gfCNCPoint2[19223] = {X 326.2725, Y 101.3575, Z -3.0000, A 0.000, B 0.000, C 0.000 }
gfCNCPoint2[19224] = {X 323.4288, Y 100.7538, Z -3.0000, A 0.000, B 0.000, C 0.000 }
gfCNCPoint2[19225] = {X 320.6373, Y 99.9425, Z -3.0000, A 0.000, B 0.000, C 0.000 }
gfCNCPoint2[19226] = {X 317.9129, Y 98.9281, Z -3.0000, A 0.000, B 0.000, C 0.000 }
gfCNCPoint2[19227] = {X 316.4064, Y 98.2325, Z -3.0000, A 0.000, B 0.000, C 0.000 }
gfCNCPoint2[19228] = {X 314.9630, Y 97.4138, Z -3.0000, A 0.000, B 0.000, C 0.000 }
gfCNCPoint2[19229] = {X 313.5930, Y 96.4776, Z -3.0000, A 0.000, B 0.000, C 0.000 }
gfCNCPoint2[19230] = {X 312.3057, Y 95.4305, Z -3.0000, A 0.000, B 0.000, C 0.000 }
gfCNCPoint2[19231] = {X 311.3087, Y 94.4389, Z -3.0000, A 0.000, B 0.000, C 0.000 }
gfCNCPoint2[19232] = {X 310.4363, Y 93.3361, Z -3.0000, A 0.000, B 0.000, C 0.000 }
gfCNCPoint2[19233] = {X 309.7010, Y 92.1376, Z -3.0000, A 0.000, B 0.000, C 0.000 }
gfCNCPoint2[19234] = {X 309.1130, Y 90.8602, Z -3.0000, A 0.000, B 0.000, C 0.000 }
gfCNCPoint2[19235] = {X 308.6807, Y 89.5222, Z -3.0000, A 0.000, B 0.000, C 0.000 }
gfCNCPoint2[19236] = {X 308.3387, Y 87.9058, Z -3.0000, A 0.000, B 0.000, C 0.000 }
gfCNCPoint2[19237] = {X 308.1366, Y 86.2660, Z -3.0000, A 0.000, B 0.000, C 0.000 }
gfCNCPoint2[19238] = {X 308.0760, Y 84.6149, Z -3.0000, A 0.000, B 0.000, C 0.000 }
gfCNCPoint2[19239] = {X 308.0773, Y 83.2310, Z -3.0000, A 0.000, B 0.000, C 0.000 }
gfCNCPoint2[19240] = {X 308.0773, Y 63.1422, Z -3.0000, A 0.000, B 0.000, C 0.000 }
gfCNCPoint2[19241] = {X 307.2288, Y 62.9475, Z -3.0000, A 0.000, B 0.000, C 0.000 }
gfCNCPoint2[19242] = {X 306.4379, Y 62.5836, Z -3.0000, A 0.000, B 0.000, C 0.000 }
gfCNCPoint2[19243] = {X 305.7380, Y 62.0658, Z -3.0000, A 0.000, B 0.000, C 0.000 }
gfCNCPoint2[19244] = {X 305.1586, Y 61.4160, Z -3.0000, A 0.000, B 0.000, C 0.000 }
gfCNCPoint2[19245] = {X 304.7241, Y 60.6616, Z -3.0000, A 0.000, B 0.000, C 0.000 }
gfCNCPoint2[19246] = {X 304.4529, Y 59.8343, Z -3.0000, A 0.000, B 0.000, C 0.000 }
gfCNCPoint2[19247] = {X 304.3564, Y 58.9691, Z -3.0000, A 0.000, B 0.000, C 0.000 }
gfCNCPoint2[19248] = {X 304.3562, Y 58.0000, Z -3.0000, A 0.000, B 0.000, C 0.000 }
gfCNCPoint2[19249] = {X 304.4625, Y 57.0565, Z -3.0000, A 0.000, B 0.000, C 0.000 }
gfCNCPoint2[19250] = {X 304.7761, Y 56.1603, Z -3.0000, A 0.000, B 0.000, C 0.000 }
gfCNCPoint2[19251] = {X 305.2813, Y 55.3564, Z -3.0000, A 0.000, B 0.000, C 0.000 }
gfCNCPoint2[19252] = {X 305.9526, Y 54.6850, Z -3.0000, A 0.000, B 0.000, C 0.000 }
gfCNCPoint2[19253] = {X 306.7566, Y 54.1799, Z -3.0000, A 0.000, B 0.000, C 0.000 }
gfCNCPoint2[19254] = {X 307.6527, Y 53.8663, Z -3.0000, A 0.000, B 0.000, C 0.000 }
gfCNCPoint2[19255] = {X 308.5962, Y 53.7600, Z -3.0000, A 0.000, B 0.000, C 0.000 }
gfCNCPoint2[19256] = {X 324.3107, Y 53.7600, Z -3.0000, A 0.000, B 0.000, C 0.000 }
gfCNCPoint2[19257] = {X 325.2542, Y 53.8663, Z -3.0000, A 0.000, B 0.000, C 0.000 }
gfCNCPoint2[19258] = {X 326.1504, Y 54.1799, Z -3.0000, A 0.000, B 0.000, C 0.000 }
gfCNCPoint2[19259] = {X 326.9543, Y 54.6850, Z -3.0000, A 0.000, B 0.000, C 0.000 }
gfCNCPoint2[19260] = {X 327.6257, Y 55.3564, Z -3.0000, A 0.000, B 0.000, C 0.000 }
gfCNCPoint2[19261] = {X 328.1308, Y 56.1603, Z -3.0000, A 0.000, B 0.000, C 0.000 }
gfCNCPoint2[19262] = {X 328.4444, Y 57.0565, Z -3.0000, A 0.000, B 0.000, C 0.000 }
gfCNCPoint2[19263] = {X 328.5507, Y 58.0000, Z -3.0000, A 0.000, B 0.000, C 0.000 }
gfCNCPoint2[19264] = {X 328.5507, Y 58.9355, Z -3.0000, A 0.000, B 0.000, C 0.000 }
gfCNCPoint2[19265] = {X 328.4560, Y 59.8053, Z -3.0000, A 0.000, B 0.000, C 0.000 }
gfCNCPoint2[19266] = {X 328.1864, Y 60.6376, Z -3.0000, A 0.000, B 0.000, C 0.000 }
gfCNCPoint2[19267] = {X 327.7532, Y 61.3977, Z -3.0000, A 0.000, B 0.000, C 0.000 }
gfCNCPoint2[19268] = {X 327.1745, Y 62.0538, Z -3.0000, A 0.000, B 0.000, C 0.000 }
gfCNCPoint2[19269] = {X 326.4744, Y 62.5785, Z -3.0000, A 0.000, B 0.000, C 0.000 }
gfCNCPoint2[19270] = {X 325.6822, Y 62.9499, Z -3.0000, A 0.000, B 0.000, C 0.000 }
gfCNCPoint2[19271] = {X 324.8311, Y 63.1523, Z -3.0000, A 0.000, B 0.000, C 0.000 }
gfCNCPoint2[19272] = {X 324.8326, Y 83.2300, Z -3.0000, A 0.000, B 0.000, C 0.000 }
gfCNCPoint2[19273] = {X 324.8461, Y 84.6151, Z -3.0000, A 0.000, B 0.000, C 0.000 }
gfCNCPoint2[19274] = {X 324.9250, Y 85.8673, Z -3.0000, A 0.000, B 0.000, C 0.000 }
gfCNCPoint2[19275] = {X 325.1520, Y 87.1014, Z -3.0000, A 0.000, B 0.000, C 0.000 }
gfCNCPoint2[19276] = {X 325.4127, Y 87.3915, Z -3.0000, A 0.000, B 0.000, C 0.000 }
gfCNCPoint2[19277] = {X 325.7358, Y 87.6100, Z -3.0000, A 0.000, B 0.000, C 0.000 }
gfCNCPoint2[19278] = {X 326.1869, Y 87.8647, Z -3.0000, A 0.000, B 0.000, C 0.000 }
gfCNCPoint2[19279] = {X 327.6340, Y 88.4662, Z -3.0000, A 0.000, B 0.000, C 0.000 }
gfCNCPoint2[19280] = {X 329.1387, Y 88.9046, Z -3.0000, A 0.000, B 0.000, C 0.000 }
gfCNCPoint2[19281] = {X 332.2202, Y 89.5215, Z -3.0000, A 0.000, B 0.000, C 0.000 }
gfCNCPoint2[19282] = {X 335.3381, Y 89.9149, Z -3.0000, A 0.000, B 0.000, C 0.000 }
gfCNCPoint2[19283] = {X 339.4788, Y 90.2356, Z -3.0000, A 0.000, B 0.000, C 0.000 }
gfCNCPoint2[19284] = {X 343.6280, Y 90.4154, Z -3.0000, A 0.000, B 0.000, C 0.000 }
gfCNCPoint2[19285] = {X 347.7809, Y 90.4540, Z -3.0000, A 0.000, B 0.000, C 0.000 }
gfCNCPoint2[19286] = {X 352.1650, Y 90.4156, Z -3.0000, A 0.000, B 0.000, C 0.000 }
gfCNCPoint2[19287] = {X 356.5449, Y 90.2196, Z -3.0000, A 0.000, B 0.000, C 0.000 }
gfCNCPoint2[19288] = {X 360.9150, Y 89.8663, Z -3.0000, A 0.000, B 0.000, C 0.000 }
gfCNCPoint2[19289] = {X 363.2338, Y 89.5779, Z -3.0000, A 0.000, B 0.000, C 0.000 }
gfCNCPoint2[19290] = {X 365.5310, Y 89.1507, Z -3.0000, A 0.000, B 0.000, C 0.000 }
gfCNCPoint2[19291] = {X 367.7985, Y 88.5862, Z -3.0000, A 0.000, B 0.000, C 0.000 }
gfCNCPoint2[19292] = {X 368.7389, Y 88.2700, Z -3.0000, A 0.000, B 0.000, C 0.000 }
gfCNCPoint2[19293] = {X 369.6379, Y 87.8503, Z -3.0000, A 0.000, B 0.000, C 0.000 }
gfCNCPoint2[19294] = {X 370.4842, Y 87.3325, Z -3.0000, A 0.000, B 0.000, C 0.000 }
gfCNCPoint2[19295] = {X 370.6562, Y 87.1535, Z -3.0000, A 0.000, B 0.000, C 0.000 }
gfCNCPoint2[19296] = {X 370.7448, Y 86.9218, Z -3.0000, A 0.000, B 0.000, C 0.000 }
gfCNCPoint2[19297] = {X 370.9367, Y 85.3801, Z -3.0000, A 0.000, B 0.000, C 0.000 }
gfCNCPoint2[19298] = {X 371.0008, Y 83.8280, Z -3.0000, A 0.000, B 0.000, C 0.000 }
gfCNCPoint2[19299] = {X 371.0008, Y 63.1422, Z -3.0000, A 0.000, B 0.000, C 0.000 }
gfCNCPoint2[19300] = {X 370.1522, Y 62.9476, Z -3.0000, A 0.000, B 0.000, C 0.000 }
gfCNCPoint2[19301] = {X 369.3612, Y 62.5838, Z -3.0000, A 0.000, B 0.000, C 0.000 }
gfCNCPoint2[19302] = {X 368.6612, Y 62.0660, Z -3.0000, A 0.000, B 0.000, C 0.000 }
gfCNCPoint2[19303] = {X 368.0817, Y 61.4162, Z -3.0000, A 0.000, B 0.000, C 0.000 }
gfCNCPoint2[19304] = {X 367.6472, Y 60.6617, Z -3.0000, A 0.000, B 0.000, C 0.000 }
gfCNCPoint2[19305] = {X 367.3760, Y 59.8344, Z -3.0000, A 0.000, B 0.000, C 0.000 }
gfCNCPoint2[19306] = {X 367.2794, Y 58.9691, Z -3.0000, A 0.000, B 0.000, C 0.000 }
gfCNCPoint2[19307] = {X 367.2793, Y 58.0000, Z -3.0000, A 0.000, B 0.000, C 0.000 }
gfCNCPoint2[19308] = {X 367.3856, Y 57.0565, Z -3.0000, A 0.000, B 0.000, C 0.000 }
gfCNCPoint2[19309] = {X 367.6992, Y 56.1603, Z -3.0000, A 0.000, B 0.000, C 0.000 }
gfCNCPoint2[19310] = {X 368.2043, Y 55.3564, Z -3.0000, A 0.000, B 0.000, C 0.000 }
gfCNCPoint2[19311] = {X 368.8757, Y 54.6850, Z -3.0000, A 0.000, B 0.000, C 0.000 }
gfCNCPoint2[19312] = {X 369.6796, Y 54.1799, Z -3.0000, A 0.000, B 0.000, C 0.000 }
gfCNCPoint2[19313] = {X 370.5758, Y 53.8663, Z -3.0000, A 0.000, B 0.000, C 0.000 }
gfCNCPoint2[19314] = {X 371.5193, Y 53.7600, Z -3.0000, A 0.000, B 0.000, C 0.000 }
gfCNCPoint2[19315] = {X 388.0597, Y 53.7600, Z -3.0000, A 0.000, B 0.000, C 0.000 }
gfCNCPoint2[19316] = {X 389.0032, Y 53.8663, Z -3.0000, A 0.000, B 0.000, C 0.000 }
gfCNCPoint2[19317] = {X 389.8993, Y 54.1799, Z -3.0000, A 0.000, B 0.000, C 0.000 }
gfCNCPoint2[19318] = {X 390.7033, Y 54.6850, Z -3.0000, A 0.000, B 0.000, C 0.000 }
gfCNCPoint2[19319] = {X 391.3746, Y 55.3564, Z -3.0000, A 0.000, B 0.000, C 0.000 }
gfCNCPoint2[19320] = {X 391.8798, Y 56.1603, Z -3.0000, A 0.000, B 0.000, C 0.000 }
gfCNCPoint2[19321] = {X 392.1934, Y 57.0565, Z -3.0000, A 0.000, B 0.000, C 0.000 }
gfCNCPoint2[19322] = {X 392.2997, Y 58.0000, Z -3.0000, A 0.000, B 0.000, C 0.000 }
gfCNCPoint2[19323] = {X 392.2997, Y 58.9342, Z -3.0000, A 0.000, B 0.000, C 0.000 }
gfCNCPoint2[19324] = {X 392.1866, Y 59.9066, Z -3.0000, A 0.000, B 0.000, C 0.000 }
gfCNCPoint2[19325] = {X 391.8536, Y 60.8272, Z -3.0000, A 0.000, B 0.000, C 0.000 }
gfCNCPoint2[19326] = {X 391.4098, Y 61.5353, Z -3.0000, A 0.000, B 0.000, C 0.000 }
gfCNCPoint2[19327] = {X 390.8364, Y 62.1431, Z -3.0000, A 0.000, B 0.000, C 0.000 }
gfCNCPoint2[19328] = {X 390.1553, Y 62.6274, Z -3.0000, A 0.000, B 0.000, C 0.000 }
gfCNCPoint2[19329] = {X 389.3929, Y 62.9695, Z -3.0000, A 0.000, B 0.000, C 0.000 }
gfCNCPoint2[19330] = {X 388.5783, Y 63.1561, Z -3.0000, A 0.000, B 0.000, C 0.000 }
gfCNCPoint2[19331] = {X 388.5763, Y 84.6150, Z -3.0000, A 0.000, B 0.000, C 0.000 }
gfCNCPoint2[19332] = {X 388.5167, Y 86.2665, Z -3.0000, A 0.000, B 0.000, C 0.000 }
gfCNCPoint2[19333] = {X 388.3133, Y 87.9065, Z -3.0000, A 0.000, B 0.000, C 0.000 }
gfCNCPoint2[19334] = {X 387.9674, Y 89.5225, Z -3.0000, A 0.000, B 0.000, C 0.000 }
gfCNCPoint2[19335] = {X 387.4388, Y 91.0992, Z -3.0000, A 0.000, B 0.000, C 0.000 }
gfCNCPoint2[19336] = {X 386.6944, Y 92.5861, Z -3.0000, A 0.000, B 0.000, C 0.000 }
gfCNCPoint2[19337] = {X 385.7486, Y 93.9539, Z -3.0000, A 0.000, B 0.000, C 0.000 }
gfCNCPoint2[19338] = {X 384.6203, Y 95.1755, Z -3.0000, A 0.000, B 0.000, C 0.000 }
gfCNCPoint2[19339] = {X 383.1126, Y 96.4458, Z -3.0000, A 0.000, B 0.000, C 0.000 }
gfCNCPoint2[19340] = {X 381.4786, Y 97.5489, Z -3.0000, A 0.000, B 0.000, C 0.000 }
gfCNCPoint2[19341] = {X 379.7367, Y 98.4723, Z -3.0000, A 0.000, B 0.000, C 0.000 }
gfCNCPoint2[19342] = {X 377.4708, Y 99.4262, Z -3.0000, A 0.000, B 0.000, C 0.000 }
gfCNCPoint2[19343] = {X 375.1422, Y 100.2147, Z -3.0000, A 0.000, B 0.000, C 0.000 }
gfCNCPoint2[19344] = {X 372.7628, Y 100.8335, Z -3.0000, A 0.000, B 0.000, C 0.000 }
gfCNCPoint2[19345] = {X 368.9550, Y 101.5702, Z -3.0000, A 0.000, B 0.000, C 0.000 }
gfCNCPoint2[19346] = {X 365.1161, Y 102.1230, Z -3.0000, A 0.000, B 0.000, C 0.000 }
gfCNCPoint2[19347] = {X 361.2551, Y 102.4906, Z -3.0000, A 0.000, B 0.000, C 0.000 }
gfCNCPoint2[19348] = {X 357.2498, Y 102.7312, Z -3.0000, A 0.000, B 0.000, C 0.000 }
gfCNCPoint2[19349] = {X 353.2403, Y 102.8846, Z -3.0000, A 0.000, B 0.000, C 0.000 }
gfCNCPoint2[19350] = {X 353.3497, Y 106.8831, Z -3.0000, A 0.000, B 0.000, C 0.000 }
gfCNCPoint2[19351] = {X 353.2381, Y 102.8046, Z -3.0000, A 0.000, B 0.000, C 0.000 }
gfCNCPoint2[19352] = {X 347.7206, Y 102.8731, Z -3.0000, A 0.000, B 0.000, C 0.000 }
gfCNCPoint2[19353] = {X 342.2035, Y 102.7764, Z -3.0000, A 0.000, B 0.000, C 0.000 }
gfCNCPoint2[19354] = {X 336.6917, Y 102.5147, Z -3.0000, A 0.000, B 0.000, C 0.000 }
gfCNCPoint2[19355] = {X 333.2080, Y 102.2391, Z -3.0000, A 0.000, B 0.000, C 0.000 }
gfCNCPoint2[19356] = {X 329.7378, Y 101.8269, Z -3.0000, A 0.000, B 0.000, C 0.000 }
gfCNCPoint2[19357] = {X 326.2865, Y 101.2787, Z -3.0000, A 0.000, B 0.000, C 0.000 }
gfCNCPoint2[19358] = {X 323.4485, Y 100.6762, Z -3.0000, A 0.000, B 0.000, C 0.000 }
gfCNCPoint2[19359] = {X 320.6624, Y 99.8666, Z -3.0000, A 0.000, B 0.000, C 0.000 }
gfCNCPoint2[19360] = {X 317.9435, Y 98.8541, Z -3.0000, A 0.000, B 0.000, C 0.000 }
gfCNCPoint2[19361] = {X 316.4430, Y 98.1614, Z -3.0000, A 0.000, B 0.000, C 0.000 }
gfCNCPoint2[19362] = {X 315.0054, Y 97.3460, Z -3.0000, A 0.000, B 0.000, C 0.000 }
gfCNCPoint2[19363] = {X 313.6408, Y 96.4135, Z -3.0000, A 0.000, B 0.000, C 0.000 }
gfCNCPoint2[19364] = {X 312.3587, Y 95.3706, Z -3.0000, A 0.000, B 0.000, C 0.000 }
gfCNCPoint2[19365] = {X 311.3684, Y 94.3857, Z -3.0000, A 0.000, B 0.000, C 0.000 }
gfCNCPoint2[19366] = {X 310.5019, Y 93.2903, Z -3.0000, A 0.000, B 0.000, C 0.000 }
gfCNCPoint2[19367] = {X 309.7715, Y 92.0999, Z -3.0000, A 0.000, B 0.000, C 0.000 }
gfCNCPoint2[19368] = {X 309.1875, Y 90.8312, Z -3.0000, A 0.000, B 0.000, C 0.000 }
gfCNCPoint2[19369] = {X 308.7582, Y 89.5022, Z -3.0000, A 0.000, B 0.000, C 0.000 }
gfCNCPoint2[19370] = {X 308.4176, Y 87.8925, Z -3.0000, A 0.000, B 0.000, C 0.000 }
gfCNCPoint2[19371] = {X 308.2164, Y 86.2595, Z -3.0000, A 0.000, B 0.000, C 0.000 }
gfCNCPoint2[19372] = {X 308.1560, Y 84.6152, Z -3.0000, A 0.000, B 0.000, C 0.000 }
gfCNCPoint2[19373] = {X 308.1573, Y 83.2311, Z -3.0000, A 0.000, B 0.000, C 0.000 }
gfCNCPoint2[19374] = {X 308.1573, Y 63.0708, Z -3.0000, A 0.000, B 0.000, C 0.000 }
gfCNCPoint2[19375] = {X 307.3120, Y 62.8909, Z -3.0000, A 0.000, B 0.000, C 0.000 }
gfCNCPoint2[19376] = {X 306.5222, Y 62.5402, Z -3.0000, A 0.000, B 0.000, C 0.000 }
gfCNCPoint2[19377] = {X 305.8219, Y 62.0338, Z -3.0000, A 0.000, B 0.000, C 0.000 }
gfCNCPoint2[19378] = {X 305.2413, Y 61.3937, Z -3.0000, A 0.000, B 0.000, C 0.000 }
gfCNCPoint2[19379] = {X 304.8054, Y 60.6474, Z -3.0000, A 0.000, B 0.000, C 0.000 }
gfCNCPoint2[19380] = {X 304.5332, Y 59.8272, Z -3.0000, A 0.000, B 0.000, C 0.000 }
gfCNCPoint2[19381] = {X 304.4364, Y 58.9684, Z -3.0000, A 0.000, B 0.000, C 0.000 }
gfCNCPoint2[19382] = {X 304.4362, Y 58.0000, Z -3.0000, A 0.000, B 0.000, C 0.000 }
gfCNCPoint2[19383] = {X 304.5405, Y 57.0743, Z -3.0000, A 0.000, B 0.000, C 0.000 }
gfCNCPoint2[19384] = {X 304.8482, Y 56.1950, Z -3.0000, A 0.000, B 0.000, C 0.000 }
gfCNCPoint2[19385] = {X 305.3438, Y 55.4063, Z -3.0000, A 0.000, B 0.000, C 0.000 }
gfCNCPoint2[19386] = {X 306.0025, Y 54.7476, Z -3.0000, A 0.000, B 0.000, C 0.000 }
gfCNCPoint2[19387] = {X 306.7913, Y 54.2520, Z -3.0000, A 0.000, B 0.000, C 0.000 }
gfCNCPoint2[19388] = {X 307.6705, Y 53.9443, Z -3.0000, A 0.000, B 0.000, C 0.000 }
gfCNCPoint2[19389] = {X 308.5962, Y 53.8400, Z -3.0000, A 0.000, B 0.000, C 0.000 }
gfCNCPoint2[19390] = {X 324.3107, Y 53.8400, Z -3.0000, A 0.000, B 0.000, C 0.000 }
gfCNCPoint2[19391] = {X 325.2364, Y 53.9443, Z -3.0000, A 0.000, B 0.000, C 0.000 }
gfCNCPoint2[19392] = {X 326.1156, Y 54.2520, Z -3.0000, A 0.000, B 0.000, C 0.000 }
gfCNCPoint2[19393] = {X 326.9044, Y 54.7476, Z -3.0000, A 0.000, B 0.000, C 0.000 }
gfCNCPoint2[19394] = {X 327.5631, Y 55.4063, Z -3.0000, A 0.000, B 0.000, C 0.000 }
gfCNCPoint2[19395] = {X 328.0587, Y 56.1950, Z -3.0000, A 0.000, B 0.000, C 0.000 }
gfCNCPoint2[19396] = {X 328.3664, Y 57.0743, Z -3.0000, A 0.000, B 0.000, C 0.000 }
gfCNCPoint2[19397] = {X 328.4707, Y 58.0000, Z -3.0000, A 0.000, B 0.000, C 0.000 }
gfCNCPoint2[19398] = {X 328.4707, Y 58.9351, Z -3.0000, A 0.000, B 0.000, C 0.000 }
gfCNCPoint2[19399] = {X 328.3757, Y 59.7983, Z -3.0000, A 0.000, B 0.000, C 0.000 }
gfCNCPoint2[19400] = {X 328.1051, Y 60.6236, Z -3.0000, A 0.000, B 0.000, C 0.000 }
gfCNCPoint2[19401] = {X 327.6706, Y 61.3756, Z -3.0000, A 0.000, B 0.000, C 0.000 }
gfCNCPoint2[19402] = {X 327.0906, Y 62.0221, Z -3.0000, A 0.000, B 0.000, C 0.000 }
gfCNCPoint2[19403] = {X 326.3901, Y 62.5354, Z -3.0000, A 0.000, B 0.000, C 0.000 }
gfCNCPoint2[19404] = {X 325.5990, Y 62.8937, Z -3.0000, A 0.000, B 0.000, C 0.000 }
gfCNCPoint2[19405] = {X 324.7510, Y 63.0816, Z -3.0000, A 0.000, B 0.000, C 0.000 }
gfCNCPoint2[19406] = {X 324.7526, Y 83.2304, Z -3.0000, A 0.000, B 0.000, C 0.000 }
gfCNCPoint2[19407] = {X 324.7661, Y 84.6154, Z -3.0000, A 0.000, B 0.000, C 0.000 }
gfCNCPoint2[19408] = {X 324.8465, Y 85.8844, Z -3.0000, A 0.000, B 0.000, C 0.000 }
gfCNCPoint2[19409] = {X 325.0779, Y 87.1348, Z -3.0000, A 0.000, B 0.000, C 0.000 }
gfCNCPoint2[19410] = {X 325.3539, Y 87.4463, Z -3.0000, A 0.000, B 0.000, C 0.000 }
gfCNCPoint2[19411] = {X 325.6979, Y 87.6805, Z -3.0000, A 0.000, B 0.000, C 0.000 }
gfCNCPoint2[19412] = {X 326.1498, Y 87.9356, Z -3.0000, A 0.000, B 0.000, C 0.000 }
gfCNCPoint2[19413] = {X 327.6062, Y 88.5412, Z -3.0000, A 0.000, B 0.000, C 0.000 }
gfCNCPoint2[19414] = {X 329.1205, Y 88.9825, Z -3.0000, A 0.000, B 0.000, C 0.000 }
gfCNCPoint2[19415] = {X 332.2075, Y 89.6005, Z -3.0000, A 0.000, B 0.000, C 0.000 }
gfCNCPoint2[19416] = {X 335.3310, Y 89.9945, Z -3.0000, A 0.000, B 0.000, C 0.000 }
gfCNCPoint2[19417] = {X 339.4742, Y 90.3155, Z -3.0000, A 0.000, B 0.000, C 0.000 }
gfCNCPoint2[19418] = {X 343.6260, Y 90.4954, Z -3.0000, A 0.000, B 0.000, C 0.000 }
gfCNCPoint2[19419] = {X 347.7815, Y 90.5340, Z -3.0000, A 0.000, B 0.000, C 0.000 }
gfCNCPoint2[19420] = {X 352.1681, Y 90.4955, Z -3.0000, A 0.000, B 0.000, C 0.000 }
gfCNCPoint2[19421] = {X 356.5504, Y 90.2994, Z -3.0000, A 0.000, B 0.000, C 0.000 }
gfCNCPoint2[19422] = {X 360.9228, Y 89.9459, Z -3.0000, A 0.000, B 0.000, C 0.000 }
gfCNCPoint2[19423] = {X 363.2463, Y 89.6569, Z -3.0000, A 0.000, B 0.000, C 0.000 }
gfCNCPoint2[19424] = {X 365.5481, Y 89.2288, Z -3.0000, A 0.000, B 0.000, C 0.000 }
gfCNCPoint2[19425] = {X 367.8201, Y 88.6632, Z -3.0000, A 0.000, B 0.000, C 0.000 }
gfCNCPoint2[19426] = {X 368.7689, Y 88.3441, Z -3.0000, A 0.000, B 0.000, C 0.000 }
gfCNCPoint2[19427] = {X 369.6759, Y 87.9207, Z -3.0000, A 0.000, B 0.000, C 0.000 }
gfCNCPoint2[19428] = {X 370.5298, Y 87.3983, Z -3.0000, A 0.000, B 0.000, C 0.000 }
gfCNCPoint2[19429] = {X 370.7237, Y 87.1964, Z -3.0000, A 0.000, B 0.000, C 0.000 }
gfCNCPoint2[19430] = {X 370.8237, Y 86.9349, Z -3.0000, A 0.000, B 0.000, C 0.000 }
gfCNCPoint2[19431] = {X 371.0164, Y 85.3867, Z -3.0000, A 0.000, B 0.000, C 0.000 }
gfCNCPoint2[19432] = {X 371.0808, Y 83.8279, Z -3.0000, A 0.000, B 0.000, C 0.000 }
gfCNCPoint2[19433] = {X 371.0808, Y 63.0709, Z -3.0000, A 0.000, B 0.000, C 0.000 }
gfCNCPoint2[19434] = {X 370.9784, Y 63.0587, Z -3.0000, A 0.000, B 0.000, C 0.000 }
gfCNCPoint2[19435] = {X 370.8762, Y 63.0441, Z -3.0000, A 0.000, B 0.000, C 0.000 }
gfCNCPoint2[19436] = {X 369.9386, Y 62.7821, Z -3.0000, A 0.000, B 0.000, C 0.000 }
gfCNCPoint2[19437] = {X 369.0876, Y 62.3093, Z -3.0000, A 0.000, B 0.000, C 0.000 }
gfCNCPoint2[19438] = {X 368.3697, Y 61.6518, Z -3.0000, A 0.000, B 0.000, C 0.000 }
gfCNCPoint2[19439] = {X 367.8243, Y 60.8454, Z -3.0000, A 0.000, B 0.000, C 0.000 }
gfCNCPoint2[19440] = {X 367.4813, Y 59.9343, Z -3.0000, A 0.000, B 0.000, C 0.000 }
gfCNCPoint2[19441] = {X 367.3594, Y 58.9684, Z -3.0000, A 0.000, B 0.000, C 0.000 }
gfCNCPoint2[19442] = {X 367.3593, Y 58.0000, Z -3.0000, A 0.000, B 0.000, C 0.000 }
gfCNCPoint2[19443] = {X 367.4636, Y 57.0743, Z -3.0000, A 0.000, B 0.000, C 0.000 }
gfCNCPoint2[19444] = {X 367.7713, Y 56.1950, Z -3.0000, A 0.000, B 0.000, C 0.000 }
gfCNCPoint2[19445] = {X 368.2669, Y 55.4063, Z -3.0000, A 0.000, B 0.000, C 0.000 }
gfCNCPoint2[19446] = {X 368.9256, Y 54.7476, Z -3.0000, A 0.000, B 0.000, C 0.000 }
gfCNCPoint2[19447] = {X 369.7143, Y 54.2520, Z -3.0000, A 0.000, B 0.000, C 0.000 }
gfCNCPoint2[19448] = {X 370.5936, Y 53.9443, Z -3.0000, A 0.000, B 0.000, C 0.000 }
gfCNCPoint2[19449] = {X 371.5193, Y 53.8400, Z -3.0000, A 0.000, B 0.000, C 0.000 }
gfCNCPoint2[19450] = {X 388.0597, Y 53.8400, Z -3.0000, A 0.000, B 0.000, C 0.000 }
gfCNCPoint2[19451] = {X 388.9854, Y 53.9443, Z -3.0000, A 0.000, B 0.000, C 0.000 }
gfCNCPoint2[19452] = {X 389.8646, Y 54.2520, Z -3.0000, A 0.000, B 0.000, C 0.000 }
gfCNCPoint2[19453] = {X 390.6534, Y 54.7476, Z -3.0000, A 0.000, B 0.000, C 0.000 }
gfCNCPoint2[19454] = {X 391.3121, Y 55.4063, Z -3.0000, A 0.000, B 0.000, C 0.000 }
gfCNCPoint2[19455] = {X 391.8077, Y 56.1950, Z -3.0000, A 0.000, B 0.000, C 0.000 }
gfCNCPoint2[19456] = {X 392.1154, Y 57.0743, Z -3.0000, A 0.000, B 0.000, C 0.000 }
gfCNCPoint2[19457] = {X 392.2197, Y 58.0000, Z -3.0000, A 0.000, B 0.000, C 0.000 }
gfCNCPoint2[19458] = {X 392.2197, Y 58.9342, Z -3.0000, A 0.000, B 0.000, C 0.000 }
gfCNCPoint2[19459] = {X 392.1088, Y 59.8883, Z -3.0000, A 0.000, B 0.000, C 0.000 }
gfCNCPoint2[19460] = {X 391.7820, Y 60.7914, Z -3.0000, A 0.000, B 0.000, C 0.000 }
gfCNCPoint2[19461] = {X 391.2381, Y 61.6189, Z -3.0000, A 0.000, B 0.000, C 0.000 }
gfCNCPoint2[19462] = {X 390.5149, Y 62.2952, Z -3.0000, A 0.000, B 0.000, C 0.000 }
gfCNCPoint2[19463] = {X 389.6528, Y 62.7826, Z -3.0000, A 0.000, B 0.000, C 0.000 }
gfCNCPoint2[19464] = {X 388.7004, Y 63.0535, Z -3.0000, A 0.000, B 0.000, C 0.000 }
gfCNCPoint2[19465] = {X 388.6002, Y 63.0683, Z -3.0000, A 0.000, B 0.000, C 0.000 }
gfCNCPoint2[19466] = {X 388.4996, Y 63.0806, Z -3.0000, A 0.000, B 0.000, C 0.000 }
gfCNCPoint2[19467] = {X 388.4963, Y 84.6154, Z -3.0000, A 0.000, B 0.000, C 0.000 }
gfCNCPoint2[19468] = {X 388.4370, Y 86.2600, Z -3.0000, A 0.000, B 0.000, C 0.000 }
gfCNCPoint2[19469] = {X 388.2344, Y 87.8931, Z -3.0000, A 0.000, B 0.000, C 0.000 }
gfCNCPoint2[19470] = {X 387.8899, Y 89.5023, Z -3.0000, A 0.000, B 0.000, C 0.000 }
gfCNCPoint2[19471] = {X 387.3650, Y 91.0684, Z -3.0000, A 0.000, B 0.000, C 0.000 }
gfCNCPoint2[19472] = {X 386.6255, Y 92.5453, Z -3.0000, A 0.000, B 0.000, C 0.000 }
gfCNCPoint2[19473] = {X 385.6862, Y 93.9039, Z -3.0000, A 0.000, B 0.000, C 0.000 }
gfCNCPoint2[19474] = {X 384.5655, Y 95.1172, Z -3.0000, A 0.000, B 0.000, C 0.000 }
gfCNCPoint2[19475] = {X 383.0643, Y 96.3820, Z -3.0000, A 0.000, B 0.000, C 0.000 }
gfCNCPoint2[19476] = {X 381.4373, Y 97.4803, Z -3.0000, A 0.000, B 0.000, C 0.000 }
gfCNCPoint2[19477] = {X 379.7030, Y 98.3998, Z -3.0000, A 0.000, B 0.000, C 0.000 }
gfCNCPoint2[19478] = {X 377.4424, Y 99.3514, Z -3.0000, A 0.000, B 0.000, C 0.000 }
gfCNCPoint2[19479] = {X 375.1192, Y 100.1380, Z -3.0000, A 0.000, B 0.000, C 0.000 }
gfCNCPoint2[19480] = {X 372.7455, Y 100.7554, Z -3.0000, A 0.000, B 0.000, C 0.000 }
gfCNCPoint2[19481] = {X 368.9415, Y 101.4914, Z -3.0000, A 0.000, B 0.000, C 0.000 }
gfCNCPoint2[19482] = {X 365.1066, Y 102.0436, Z -3.0000, A 0.000, B 0.000, C 0.000 }
gfCNCPoint2[19483] = {X 361.2495, Y 102.4108, Z -3.0000, A 0.000, B 0.000, C 0.000 }
gfCNCPoint2[19484] = {X 357.2459, Y 102.6513, Z -3.0000, A 0.000, B 0.000, C 0.000 }
gfCNCPoint2[19485] = {X 353.2381, Y 102.8046, Z -3.0000, A 0.000, B 0.000, C 0.000 }
gfCNCPoint2[19486] = {X 353.3475, Y 106.8031, Z -3.0000, A 0.000, B 0.000, C 0.000 }
gfCNCPoint2[19487] = {X 353.2359, Y 102.7246, Z -3.0000, A 0.000, B 0.000, C 0.000 }
gfCNCPoint2[19488] = {X 347.7207, Y 102.7931, Z -3.0000, A 0.000, B 0.000, C 0.000 }
gfCNCPoint2[19489] = {X 342.2060, Y 102.6965, Z -3.0000, A 0.000, B 0.000, C 0.000 }
gfCNCPoint2[19490] = {X 336.6967, Y 102.4349, Z -3.0000, A 0.000, B 0.000, C 0.000 }
gfCNCPoint2[19491] = {X 333.2160, Y 102.1595, Z -3.0000, A 0.000, B 0.000, C 0.000 }
gfCNCPoint2[19492] = {X 329.7488, Y 101.7477, Z -3.0000, A 0.000, B 0.000, C 0.000 }
gfCNCPoint2[19493] = {X 326.3004, Y 101.1999, Z -3.0000, A 0.000, B 0.000, C 0.000 }
gfCNCPoint2[19494] = {X 323.4680, Y 100.5987, Z -3.0000, A 0.000, B 0.000, C 0.000 }
gfCNCPoint2[19495] = {X 320.6875, Y 99.7906, Z -3.0000, A 0.000, B 0.000, C 0.000 }
gfCNCPoint2[19496] = {X 317.9740, Y 98.7802, Z -3.0000, A 0.000, B 0.000, C 0.000 }
gfCNCPoint2[19497] = {X 316.4795, Y 98.0902, Z -3.0000, A 0.000, B 0.000, C 0.000 }
gfCNCPoint2[19498] = {X 315.0478, Y 97.2781, Z -3.0000, A 0.000, B 0.000, C 0.000 }
gfCNCPoint2[19499] = {X 313.6887, Y 96.3494, Z -3.0000, A 0.000, B 0.000, C 0.000 }
gfCNCPoint2[19500] = {X 312.4117, Y 95.3107, Z -3.0000, A 0.000, B 0.000, C 0.000 }
gfCNCPoint2[19501] = {X 311.4282, Y 94.3325, Z -3.0000, A 0.000, B 0.000, C 0.000 }
gfCNCPoint2[19502] = {X 310.5676, Y 93.2446, Z -3.0000, A 0.000, B 0.000, C 0.000 }
gfCNCPoint2[19503] = {X 309.8421, Y 92.0622, Z -3.0000, A 0.000, B 0.000, C 0.000 }
gfCNCPoint2[19504] = {X 309.2621, Y 90.8021, Z -3.0000, A 0.000, B 0.000, C 0.000 }
gfCNCPoint2[19505] = {X 308.8356, Y 89.4821, Z -3.0000, A 0.000, B 0.000, C 0.000 }
gfCNCPoint2[19506] = {X 308.4965, Y 87.8791, Z -3.0000, A 0.000, B 0.000, C 0.000 }
gfCNCPoint2[19507] = {X 308.2961, Y 86.2529, Z -3.0000, A 0.000, B 0.000, C 0.000 }
gfCNCPoint2[19508] = {X 308.2360, Y 84.6155, Z -3.0000, A 0.000, B 0.000, C 0.000 }
gfCNCPoint2[19509] = {X 308.2373, Y 83.2312, Z -3.0000, A 0.000, B 0.000, C 0.000 }
gfCNCPoint2[19510] = {X 308.2373, Y 62.9982, Z -3.0000, A 0.000, B 0.000, C 0.000 }
gfCNCPoint2[19511] = {X 307.3955, Y 62.8334, Z -3.0000, A 0.000, B 0.000, C 0.000 }
gfCNCPoint2[19512] = {X 306.6068, Y 62.4961, Z -3.0000, A 0.000, B 0.000, C 0.000 }
gfCNCPoint2[19513] = {X 305.9060, Y 62.0015, Z -3.0000, A 0.000, B 0.000, C 0.000 }
gfCNCPoint2[19514] = {X 305.3241, Y 61.3712, Z -3.0000, A 0.000, B 0.000, C 0.000 }
gfCNCPoint2[19515] = {X 304.8868, Y 60.6332, Z -3.0000, A 0.000, B 0.000, C 0.000 }
gfCNCPoint2[19516] = {X 304.6136, Y 59.8200, Z -3.0000, A 0.000, B 0.000, C 0.000 }
gfCNCPoint2[19517] = {X 304.5164, Y 58.9678, Z -3.0000, A 0.000, B 0.000, C 0.000 }
gfCNCPoint2[19518] = {X 304.5162, Y 58.0000, Z -3.0000, A 0.000, B 0.000, C 0.000 }
gfCNCPoint2[19519] = {X 304.6185, Y 57.0921, Z -3.0000, A 0.000, B 0.000, C 0.000 }
gfCNCPoint2[19520] = {X 304.9203, Y 56.2298, Z -3.0000, A 0.000, B 0.000, C 0.000 }
gfCNCPoint2[19521] = {X 305.4064, Y 55.4562, Z -3.0000, A 0.000, B 0.000, C 0.000 }
gfCNCPoint2[19522] = {X 306.0524, Y 54.8101, Z -3.0000, A 0.000, B 0.000, C 0.000 }
gfCNCPoint2[19523] = {X 306.8260, Y 54.3240, Z -3.0000, A 0.000, B 0.000, C 0.000 }
gfCNCPoint2[19524] = {X 307.6883, Y 54.0223, Z -3.0000, A 0.000, B 0.000, C 0.000 }
gfCNCPoint2[19525] = {X 308.5962, Y 53.9200, Z -3.0000, A 0.000, B 0.000, C 0.000 }
gfCNCPoint2[19526] = {X 324.3107, Y 53.9200, Z -3.0000, A 0.000, B 0.000, C 0.000 }
gfCNCPoint2[19527] = {X 325.2186, Y 54.0223, Z -3.0000, A 0.000, B 0.000, C 0.000 }
gfCNCPoint2[19528] = {X 326.0809, Y 54.3240, Z -3.0000, A 0.000, B 0.000, C 0.000 }
gfCNCPoint2[19529] = {X 326.8545, Y 54.8101, Z -3.0000, A 0.000, B 0.000, C 0.000 }
gfCNCPoint2[19530] = {X 327.5006, Y 55.4562, Z -3.0000, A 0.000, B 0.000, C 0.000 }
gfCNCPoint2[19531] = {X 327.9866, Y 56.2298, Z -3.0000, A 0.000, B 0.000, C 0.000 }
gfCNCPoint2[19532] = {X 328.2884, Y 57.0921, Z -3.0000, A 0.000, B 0.000, C 0.000 }
gfCNCPoint2[19533] = {X 328.3907, Y 58.0000, Z -3.0000, A 0.000, B 0.000, C 0.000 }
gfCNCPoint2[19534] = {X 328.3907, Y 58.9346, Z -3.0000, A 0.000, B 0.000, C 0.000 }
gfCNCPoint2[19535] = {X 328.2953, Y 59.7914, Z -3.0000, A 0.000, B 0.000, C 0.000 }
gfCNCPoint2[19536] = {X 328.0237, Y 60.6095, Z -3.0000, A 0.000, B 0.000, C 0.000 }
gfCNCPoint2[19537] = {X 327.5878, Y 61.3533, Z -3.0000, A 0.000, B 0.000, C 0.000 }
gfCNCPoint2[19538] = {X 327.0066, Y 61.9900, Z -3.0000, A 0.000, B 0.000, C 0.000 }
gfCNCPoint2[19539] = {X 326.3057, Y 62.4918, Z -3.0000, A 0.000, B 0.000, C 0.000 }
gfCNCPoint2[19540] = {X 325.5156, Y 62.8367, Z -3.0000, A 0.000, B 0.000, C 0.000 }
gfCNCPoint2[19541] = {X 324.6710, Y 63.0096, Z -3.0000, A 0.000, B 0.000, C 0.000 }
gfCNCPoint2[19542] = {X 324.6726, Y 83.2309, Z -3.0000, A 0.000, B 0.000, C 0.000 }
gfCNCPoint2[19543] = {X 324.6861, Y 84.6156, Z -3.0000, A 0.000, B 0.000, C 0.000 }
gfCNCPoint2[19544] = {X 324.7680, Y 85.9014, Z -3.0000, A 0.000, B 0.000, C 0.000 }
gfCNCPoint2[19545] = {X 325.0037, Y 87.1680, Z -3.0000, A 0.000, B 0.000, C 0.000 }
gfCNCPoint2[19546] = {X 325.2949, Y 87.5009, Z -3.0000, A 0.000, B 0.000, C 0.000 }
gfCNCPoint2[19547] = {X 325.6599, Y 87.7509, Z -3.0000, A 0.000, B 0.000, C 0.000 }
gfCNCPoint2[19548] = {X 326.1127, Y 88.0066, Z -3.0000, A 0.000, B 0.000, C 0.000 }
gfCNCPoint2[19549] = {X 327.5784, Y 88.6162, Z -3.0000, A 0.000, B 0.000, C 0.000 }
gfCNCPoint2[19550] = {X 329.1024, Y 89.0604, Z -3.0000, A 0.000, B 0.000, C 0.000 }
gfCNCPoint2[19551] = {X 332.1948, Y 89.6795, Z -3.0000, A 0.000, B 0.000, C 0.000 }
gfCNCPoint2[19552] = {X 335.3238, Y 90.0742, Z -3.0000, A 0.000, B 0.000, C 0.000 }
gfCNCPoint2[19553] = {X 339.4695, Y 90.3953, Z -3.0000, A 0.000, B 0.000, C 0.000 }
gfCNCPoint2[19554] = {X 343.6236, Y 90.5753, Z -3.0000, A 0.000, B 0.000, C 0.000 }
gfCNCPoint2[19555] = {X 347.7815, Y 90.6140, Z -3.0000, A 0.000, B 0.000, C 0.000 }
gfCNCPoint2[19556] = {X 352.1706, Y 90.5755, Z -3.0000, A 0.000, B 0.000, C 0.000 }
gfCNCPoint2[19557] = {X 356.5556, Y 90.3792, Z -3.0000, A 0.000, B 0.000, C 0.000 }
gfCNCPoint2[19558] = {X 360.9307, Y 90.0255, Z -3.0000, A 0.000, B 0.000, C 0.000 }
gfCNCPoint2[19559] = {X 363.2588, Y 89.7359, Z -3.0000, A 0.000, B 0.000, C 0.000 }
gfCNCPoint2[19560] = {X 365.5653, Y 89.3070, Z -3.0000, A 0.000, B 0.000, C 0.000 }
gfCNCPoint2[19561] = {X 367.8418, Y 88.7402, Z -3.0000, A 0.000, B 0.000, C 0.000 }
gfCNCPoint2[19562] = {X 368.7989, Y 88.4183, Z -3.0000, A 0.000, B 0.000, C 0.000 }
gfCNCPoint2[19563] = {X 369.7139, Y 87.9911, Z -3.0000, A 0.000, B 0.000, C 0.000 }
gfCNCPoint2[19564] = {X 370.5753, Y 87.4640, Z -3.0000, A 0.000, B 0.000, C 0.000 }
gfCNCPoint2[19565] = {X 370.7913, Y 87.2392, Z -3.0000, A 0.000, B 0.000, C 0.000 }
gfCNCPoint2[19566] = {X 370.9026, Y 86.9481, Z -3.0000, A 0.000, B 0.000, C 0.000 }
gfCNCPoint2[19567] = {X 371.0962, Y 85.3933, Z -3.0000, A 0.000, B 0.000, C 0.000 }
gfCNCPoint2[19568] = {X 371.1608, Y 83.8279, Z -3.0000, A 0.000, B 0.000, C 0.000 }
gfCNCPoint2[19569] = {X 371.1608, Y 62.9983, Z -3.0000, A 0.000, B 0.000, C 0.000 }
gfCNCPoint2[19570] = {X 371.0244, Y 62.9839, Z -3.0000, A 0.000, B 0.000, C 0.000 }
gfCNCPoint2[19571] = {X 370.8886, Y 62.9650, Z -3.0000, A 0.000, B 0.000, C 0.000 }
gfCNCPoint2[19572] = {X 369.9690, Y 62.7081, Z -3.0000, A 0.000, B 0.000, C 0.000 }
gfCNCPoint2[19573] = {X 369.1344, Y 62.2444, Z -3.0000, A 0.000, B 0.000, C 0.000 }
gfCNCPoint2[19574] = {X 368.4303, Y 61.5995, Z -3.0000, A 0.000, B 0.000, C 0.000 }
gfCNCPoint2[19575] = {X 367.8954, Y 60.8086, Z -3.0000, A 0.000, B 0.000, C 0.000 }
gfCNCPoint2[19576] = {X 367.5590, Y 59.9150, Z -3.0000, A 0.000, B 0.000, C 0.000 }
gfCNCPoint2[19577] = {X 367.4394, Y 58.9678, Z -3.0000, A 0.000, B 0.000, C 0.000 }
gfCNCPoint2[19578] = {X 367.4393, Y 58.0000, Z -3.0000, A 0.000, B 0.000, C 0.000 }
gfCNCPoint2[19579] = {X 367.5416, Y 57.0921, Z -3.0000, A 0.000, B 0.000, C 0.000 }
gfCNCPoint2[19580] = {X 367.8433, Y 56.2298, Z -3.0000, A 0.000, B 0.000, C 0.000 }
gfCNCPoint2[19581] = {X 368.3294, Y 55.4562, Z -3.0000, A 0.000, B 0.000, C 0.000 }
gfCNCPoint2[19582] = {X 368.9754, Y 54.8101, Z -3.0000, A 0.000, B 0.000, C 0.000 }
gfCNCPoint2[19583] = {X 369.7490, Y 54.3240, Z -3.0000, A 0.000, B 0.000, C 0.000 }
gfCNCPoint2[19584] = {X 370.6114, Y 54.0223, Z -3.0000, A 0.000, B 0.000, C 0.000 }
gfCNCPoint2[19585] = {X 371.5193, Y 53.9200, Z -3.0000, A 0.000, B 0.000, C 0.000 }
gfCNCPoint2[19586] = {X 388.0597, Y 53.9200, Z -3.0000, A 0.000, B 0.000, C 0.000 }
gfCNCPoint2[19587] = {X 388.9676, Y 54.0223, Z -3.0000, A 0.000, B 0.000, C 0.000 }
gfCNCPoint2[19588] = {X 389.8299, Y 54.3240, Z -3.0000, A 0.000, B 0.000, C 0.000 }
gfCNCPoint2[19589] = {X 390.6035, Y 54.8101, Z -3.0000, A 0.000, B 0.000, C 0.000 }
gfCNCPoint2[19590] = {X 391.2496, Y 55.4562, Z -3.0000, A 0.000, B 0.000, C 0.000 }
gfCNCPoint2[19591] = {X 391.7356, Y 56.2298, Z -3.0000, A 0.000, B 0.000, C 0.000 }
gfCNCPoint2[19592] = {X 392.0374, Y 57.0921, Z -3.0000, A 0.000, B 0.000, C 0.000 }
gfCNCPoint2[19593] = {X 392.1397, Y 58.0000, Z -3.0000, A 0.000, B 0.000, C 0.000 }
gfCNCPoint2[19594] = {X 392.1397, Y 58.9342, Z -3.0000, A 0.000, B 0.000, C 0.000 }
gfCNCPoint2[19595] = {X 392.0309, Y 59.8699, Z -3.0000, A 0.000, B 0.000, C 0.000 }
gfCNCPoint2[19596] = {X 391.7104, Y 60.7557, Z -3.0000, A 0.000, B 0.000, C 0.000 }
gfCNCPoint2[19597] = {X 391.1769, Y 61.5673, Z -3.0000, A 0.000, B 0.000, C 0.000 }
gfCNCPoint2[19598] = {X 390.4675, Y 62.2308, Z -3.0000, A 0.000, B 0.000, C 0.000 }
gfCNCPoint2[19599] = {X 389.6220, Y 62.7087, Z -3.0000, A 0.000, B 0.000, C 0.000 }
gfCNCPoint2[19600] = {X 388.6878, Y 62.9745, Z -3.0000, A 0.000, B 0.000, C 0.000 }
gfCNCPoint2[19601] = {X 388.5546, Y 62.9936, Z -3.0000, A 0.000, B 0.000, C 0.000 }
gfCNCPoint2[19602] = {X 388.4208, Y 63.0082, Z -3.0000, A 0.000, B 0.000, C 0.000 }
gfCNCPoint2[19603] = {X 388.4183, Y 63.1547, Z -3.0000, A 0.000, B 0.000, C 0.000 }
gfCNCPoint2[19604] = {X 388.4163, Y 84.6157, Z -3.0000, A 0.000, B 0.000, C 0.000 }
gfCNCPoint2[19605] = {X 388.3573, Y 86.2535, Z -3.0000, A 0.000, B 0.000, C 0.000 }
gfCNCPoint2[19606] = {X 388.1555, Y 87.8798, Z -3.0000, A 0.000, B 0.000, C 0.000 }
gfCNCPoint2[19607] = {X 387.8125, Y 89.4823, Z -3.0000, A 0.000, B 0.000, C 0.000 }
gfCNCPoint2[19608] = {X 387.2911, Y 91.0377, Z -3.0000, A 0.000, B 0.000, C 0.000 }
gfCNCPoint2[19609] = {X 386.5567, Y 92.5045, Z -3.0000, A 0.000, B 0.000, C 0.000 }
gfCNCPoint2[19610] = {X 385.6238, Y 93.8538, Z -3.0000, A 0.000, B 0.000, C 0.000 }
gfCNCPoint2[19611] = {X 384.5107, Y 95.0589, Z -3.0000, A 0.000, B 0.000, C 0.000 }
gfCNCPoint2[19612] = {X 383.0160, Y 96.3182, Z -3.0000, A 0.000, B 0.000, C 0.000 }
gfCNCPoint2[19613] = {X 381.3961, Y 97.4117, Z -3.0000, A 0.000, B 0.000, C 0.000 }
gfCNCPoint2[19614] = {X 379.6693, Y 98.3272, Z -3.0000, A 0.000, B 0.000, C 0.000 }
gfCNCPoint2[19615] = {X 377.4141, Y 99.2766, Z -3.0000, A 0.000, B 0.000, C 0.000 }
gfCNCPoint2[19616] = {X 375.0963, Y 100.0614, Z -3.0000, A 0.000, B 0.000, C 0.000 }
gfCNCPoint2[19617] = {X 372.7282, Y 100.6773, Z -3.0000, A 0.000, B 0.000, C 0.000 }
gfCNCPoint2[19618] = {X 368.9280, Y 101.4125, Z -3.0000, A 0.000, B 0.000, C 0.000 }
gfCNCPoint2[19619] = {X 365.0970, Y 101.9641, Z -3.0000, A 0.000, B 0.000, C 0.000 }
gfCNCPoint2[19620] = {X 361.2438, Y 102.3310, Z -3.0000, A 0.000, B 0.000, C 0.000 }
gfCNCPoint2[19621] = {X 357.2420, Y 102.5713, Z -3.0000, A 0.000, B 0.000, C 0.000 }
gfCNCPoint2[19622] = {X 353.2359, Y 102.7246, Z -3.0000, A 0.000, B 0.000, C 0.000 }
gfCNCPoint2[19623] = {X 353.3453, Y 106.7231, Z -3.0000, A 0.000, B 0.000, C 0.000 }
gfCNCPoint2[19624] = {X 353.2337, Y 102.6447, Z -3.0000, A 0.000, B 0.000, C 0.000 }
gfCNCPoint2[19625] = {X 347.7209, Y 102.7131, Z -3.0000, A 0.000, B 0.000, C 0.000 }
gfCNCPoint2[19626] = {X 342.2086, Y 102.6165, Z -3.0000, A 0.000, B 0.000, C 0.000 }
gfCNCPoint2[19627] = {X 336.7017, Y 102.3550, Z -3.0000, A 0.000, B 0.000, C 0.000 }
gfCNCPoint2[19628] = {X 333.2240, Y 102.0799, Z -3.0000, A 0.000, B 0.000, C 0.000 }
gfCNCPoint2[19629] = {X 329.7598, Y 101.6684, Z -3.0000, A 0.000, B 0.000, C 0.000 }
gfCNCPoint2[19630] = {X 326.3144, Y 101.1212, Z -3.0000, A 0.000, B 0.000, C 0.000 }
gfCNCPoint2[19631] = {X 323.4876, Y 100.5211, Z -3.0000, A 0.000, B 0.000, C 0.000 }
gfCNCPoint2[19632] = {X 320.7127, Y 99.7147, Z -3.0000, A 0.000, B 0.000, C 0.000 }
gfCNCPoint2[19633] = {X 318.0046, Y 98.7063, Z -3.0000, A 0.000, B 0.000, C 0.000 }
gfCNCPoint2[19634] = {X 316.5161, Y 98.0191, Z -3.0000, A 0.000, B 0.000, C 0.000 }
gfCNCPoint2[19635] = {X 315.0901, Y 97.2102, Z -3.0000, A 0.000, B 0.000, C 0.000 }
gfCNCPoint2[19636] = {X 313.7365, Y 96.2853, Z -3.0000, A 0.000, B 0.000, C 0.000 }
gfCNCPoint2[19637] = {X 312.4647, Y 95.2507, Z -3.0000, A 0.000, B 0.000, C 0.000 }
gfCNCPoint2[19638] = {X 311.4879, Y 94.2793, Z -3.0000, A 0.000, B 0.000, C 0.000 }
gfCNCPoint2[19639] = {X 310.6332, Y 93.1988, Z -3.0000, A 0.000, B 0.000, C 0.000 }
gfCNCPoint2[19640] = {X 309.9127, Y 92.0245, Z -3.0000, A 0.000, B 0.000, C 0.000 }
gfCNCPoint2[19641] = {X 309.3366, Y 90.7731, Z -3.0000, A 0.000, B 0.000, C 0.000 }
gfCNCPoint2[19642] = {X 308.9131, Y 89.4621, Z -3.0000, A 0.000, B 0.000, C 0.000 }
gfCNCPoint2[19643] = {X 308.5754, Y 87.8658, Z -3.0000, A 0.000, B 0.000, C 0.000 }
gfCNCPoint2[19644] = {X 308.3759, Y 86.2464, Z -3.0000, A 0.000, B 0.000, C 0.000 }
gfCNCPoint2[19645] = {X 308.3160, Y 84.6159, Z -3.0000, A 0.000, B 0.000, C 0.000 }
gfCNCPoint2[19646] = {X 308.3173, Y 83.2313, Z -3.0000, A 0.000, B 0.000, C 0.000 }
gfCNCPoint2[19647] = {X 308.3173, Y 62.9243, Z -3.0000, A 0.000, B 0.000, C 0.000 }
gfCNCPoint2[19648] = {X 307.4746, Y 62.7736, Z -3.0000, A 0.000, B 0.000, C 0.000 }
gfCNCPoint2[19649] = {X 306.6833, Y 62.4470, Z -3.0000, A 0.000, B 0.000, C 0.000 }
gfCNCPoint2[19650] = {X 305.9796, Y 61.9595, Z -3.0000, A 0.000, B 0.000, C 0.000 }
gfCNCPoint2[19651] = {X 305.3957, Y 61.3334, Z -3.0000, A 0.000, B 0.000, C 0.000 }
gfCNCPoint2[19652] = {X 304.9585, Y 60.5974, Z -3.0000, A 0.000, B 0.000, C 0.000 }
gfCNCPoint2[19653] = {X 304.6878, Y 59.7852, Z -3.0000, A 0.000, B 0.000, C 0.000 }
gfCNCPoint2[19654] = {X 304.5962, Y 58.9340, Z -3.0000, A 0.000, B 0.000, C 0.000 }
gfCNCPoint2[19655] = {X 304.5962, Y 58.0000, Z -3.0000, A 0.000, B 0.000, C 0.000 }
gfCNCPoint2[19656] = {X 304.6965, Y 57.1099, Z -3.0000, A 0.000, B 0.000, C 0.000 }
gfCNCPoint2[19657] = {X 304.9923, Y 56.2645, Z -3.0000, A 0.000, B 0.000, C 0.000 }
gfCNCPoint2[19658] = {X 305.4689, Y 55.5060, Z -3.0000, A 0.000, B 0.000, C 0.000 }
gfCNCPoint2[19659] = {X 306.1023, Y 54.8727, Z -3.0000, A 0.000, B 0.000, C 0.000 }
gfCNCPoint2[19660] = {X 306.8607, Y 54.3961, Z -3.0000, A 0.000, B 0.000, C 0.000 }
gfCNCPoint2[19661] = {X 307.7061, Y 54.1003, Z -3.0000, A 0.000, B 0.000, C 0.000 }
gfCNCPoint2[19662] = {X 308.5962, Y 54.0000, Z -3.0000, A 0.000, B 0.000, C 0.000 }
gfCNCPoint2[19663] = {X 324.3107, Y 54.0000, Z -3.0000, A 0.000, B 0.000, C 0.000 }
gfCNCPoint2[19664] = {X 325.2008, Y 54.1003, Z -3.0000, A 0.000, B 0.000, C 0.000 }
gfCNCPoint2[19665] = {X 326.0462, Y 54.3961, Z -3.0000, A 0.000, B 0.000, C 0.000 }
gfCNCPoint2[19666] = {X 326.8046, Y 54.8727, Z -3.0000, A 0.000, B 0.000, C 0.000 }
gfCNCPoint2[19667] = {X 327.4380, Y 55.5060, Z -3.0000, A 0.000, B 0.000, C 0.000 }
gfCNCPoint2[19668] = {X 327.9146, Y 56.2645, Z -3.0000, A 0.000, B 0.000, C 0.000 }
gfCNCPoint2[19669] = {X 328.2104, Y 57.1099, Z -3.0000, A 0.000, B 0.000, C 0.000 }
gfCNCPoint2[19670] = {X 328.3107, Y 58.0000, Z -3.0000, A 0.000, B 0.000, C 0.000 }
gfCNCPoint2[19671] = {X 328.3107, Y 58.9341, Z -3.0000, A 0.000, B 0.000, C 0.000 }
gfCNCPoint2[19672] = {X 328.2149, Y 59.7844, Z -3.0000, A 0.000, B 0.000, C 0.000 }
gfCNCPoint2[19673] = {X 327.9423, Y 60.5954, Z -3.0000, A 0.000, B 0.000, C 0.000 }
gfCNCPoint2[19674] = {X 327.5049, Y 61.3308, Z -3.0000, A 0.000, B 0.000, C 0.000 }
gfCNCPoint2[19675] = {X 326.9224, Y 61.9575, Z -3.0000, A 0.000, B 0.000, C 0.000 }
gfCNCPoint2[19676] = {X 326.2209, Y 62.4475, Z -3.0000, A 0.000, B 0.000, C 0.000 }
gfCNCPoint2[19677] = {X 325.4320, Y 62.7788, Z -3.0000, A 0.000, B 0.000, C 0.000 }
gfCNCPoint2[19678] = {X 324.5910, Y 62.9364, Z -3.0000, A 0.000, B 0.000, C 0.000 }
gfCNCPoint2[19679] = {X 324.5926, Y 83.2313, Z -3.0000, A 0.000, B 0.000, C 0.000 }
gfCNCPoint2[19680] = {X 324.6061, Y 84.6159, Z -3.0000, A 0.000, B 0.000, C 0.000 }
gfCNCPoint2[19681] = {X 324.6894, Y 85.9182, Z -3.0000, A 0.000, B 0.000, C 0.000 }
gfCNCPoint2[19682] = {X 324.9294, Y 87.2009, Z -3.0000, A 0.000, B 0.000, C 0.000 }
gfCNCPoint2[19683] = {X 325.2359, Y 87.5555, Z -3.0000, A 0.000, B 0.000, C 0.000 }
gfCNCPoint2[19684] = {X 325.6219, Y 87.8213, Z -3.0000, A 0.000, B 0.000, C 0.000 }
gfCNCPoint2[19685] = {X 326.0756, Y 88.0775, Z -3.0000, A 0.000, B 0.000, C 0.000 }
gfCNCPoint2[19686] = {X 327.5506, Y 88.6912, Z -3.0000, A 0.000, B 0.000, C 0.000 }
gfCNCPoint2[19687] = {X 329.0843, Y 89.1383, Z -3.0000, A 0.000, B 0.000, C 0.000 }
gfCNCPoint2[19688] = {X 332.1822, Y 89.7585, Z -3.0000, A 0.000, B 0.000, C 0.000 }
gfCNCPoint2[19689] = {X 335.3167, Y 90.1539, Z -3.0000, A 0.000, B 0.000, C 0.000 }
gfCNCPoint2[19690] = {X 339.4647, Y 90.4752, Z -3.0000, A 0.000, B 0.000, C 0.000 }
gfCNCPoint2[19691] = {X 343.6212, Y 90.6553, Z -3.0000, A 0.000, B 0.000, C 0.000 }
gfCNCPoint2[19692] = {X 347.7814, Y 90.6940, Z -3.0000, A 0.000, B 0.000, C 0.000 }
gfCNCPoint2[19693] = {X 352.1732, Y 90.6554, Z -3.0000, A 0.000, B 0.000, C 0.000 }
gfCNCPoint2[19694] = {X 356.5609, Y 90.4591, Z -3.0000, A 0.000, B 0.000, C 0.000 }
gfCNCPoint2[19695] = {X 360.9386, Y 90.1052, Z -3.0000, A 0.000, B 0.000, C 0.000 }
gfCNCPoint2[19696] = {X 363.2713, Y 89.8150, Z -3.0000, A 0.000, B 0.000, C 0.000 }
gfCNCPoint2[19697] = {X 365.5824, Y 89.3851, Z -3.0000, A 0.000, B 0.000, C 0.000 }
gfCNCPoint2[19698] = {X 367.8634, Y 88.8172, Z -3.0000, A 0.000, B 0.000, C 0.000 }
gfCNCPoint2[19699] = {X 368.8289, Y 88.4924, Z -3.0000, A 0.000, B 0.000, C 0.000 }
gfCNCPoint2[19700] = {X 369.7519, Y 88.0615, Z -3.0000, A 0.000, B 0.000, C 0.000 }
gfCNCPoint2[19701] = {X 370.6208, Y 87.5298, Z -3.0000, A 0.000, B 0.000, C 0.000 }
gfCNCPoint2[19702] = {X 370.8588, Y 87.2821, Z -3.0000, A 0.000, B 0.000, C 0.000 }
gfCNCPoint2[19703] = {X 370.9815, Y 86.9612, Z -3.0000, A 0.000, B 0.000, C 0.000 }
gfCNCPoint2[19704] = {X 371.1759, Y 85.3999, Z -3.0000, A 0.000, B 0.000, C 0.000 }
gfCNCPoint2[19705] = {X 371.2408, Y 83.8279, Z -3.0000, A 0.000, B 0.000, C 0.000 }
gfCNCPoint2[19706] = {X 371.2391, Y 63.0388, Z -3.0000, A 0.000, B 0.000, C 0.000 }
gfCNCPoint2[19707] = {X 371.2440, Y 62.9246, Z -3.0000, A 0.000, B 0.000, C 0.000 }
gfCNCPoint2[19708] = {X 371.0721, Y 62.9090, Z -3.0000, A 0.000, B 0.000, C 0.000 }
gfCNCPoint2[19709] = {X 370.9010, Y 62.8860, Z -3.0000, A 0.000, B 0.000, C 0.000 }
gfCNCPoint2[19710] = {X 369.9943, Y 62.6320, Z -3.0000, A 0.000, B 0.000, C 0.000 }
gfCNCPoint2[19711] = {X 369.1722, Y 62.1731, Z -3.0000, A 0.000, B 0.000, C 0.000 }
gfCNCPoint2[19712] = {X 368.4801, Y 61.5347, Z -3.0000, A 0.000, B 0.000, C 0.000 }
gfCNCPoint2[19713] = {X 367.9564, Y 60.7523, Z -3.0000, A 0.000, B 0.000, C 0.000 }
gfCNCPoint2[19714] = {X 367.6301, Y 59.8691, Z -3.0000, A 0.000, B 0.000, C 0.000 }
gfCNCPoint2[19715] = {X 367.5193, Y 58.9340, Z -3.0000, A 0.000, B 0.000, C 0.000 }
gfCNCPoint2[19716] = {X 367.5193, Y 58.0000, Z -3.0000, A 0.000, B 0.000, C 0.000 }
gfCNCPoint2[19717] = {X 367.6196, Y 57.1099, Z -3.0000, A 0.000, B 0.000, C 0.000 }
gfCNCPoint2[19718] = {X 367.9154, Y 56.2645, Z -3.0000, A 0.000, B 0.000, C 0.000 }
gfCNCPoint2[19719] = {X 368.3920, Y 55.5060, Z -3.0000, A 0.000, B 0.000, C 0.000 }
gfCNCPoint2[19720] = {X 369.0253, Y 54.8727, Z -3.0000, A 0.000, B 0.000, C 0.000 }
gfCNCPoint2[19721] = {X 369.7837, Y 54.3961, Z -3.0000, A 0.000, B 0.000, C 0.000 }
gfCNCPoint2[19722] = {X 370.6292, Y 54.1003, Z -3.0000, A 0.000, B 0.000, C 0.000 }
gfCNCPoint2[19723] = {X 371.5193, Y 54.0000, Z -3.0000, A 0.000, B 0.000, C 0.000 }
gfCNCPoint2[19724] = {X 388.0597, Y 54.0000, Z -3.0000, A 0.000, B 0.000, C 0.000 }
gfCNCPoint2[19725] = {X 388.9498, Y 54.1003, Z -3.0000, A 0.000, B 0.000, C 0.000 }
gfCNCPoint2[19726] = {X 389.7952, Y 54.3961, Z -3.0000, A 0.000, B 0.000, C 0.000 }
gfCNCPoint2[19727] = {X 390.5536, Y 54.8727, Z -3.0000, A 0.000, B 0.000, C 0.000 }
gfCNCPoint2[19728] = {X 391.1870, Y 55.5060, Z -3.0000, A 0.000, B 0.000, C 0.000 }
gfCNCPoint2[19729] = {X 391.6636, Y 56.2645, Z -3.0000, A 0.000, B 0.000, C 0.000 }
gfCNCPoint2[19730] = {X 391.9594, Y 57.1099, Z -3.0000, A 0.000, B 0.000, C 0.000 }
gfCNCPoint2[19731] = {X 392.0597, Y 58.0000, Z -3.0000, A 0.000, B 0.000, C 0.000 }
gfCNCPoint2[19732] = {X 392.0595, Y 58.9671, Z -3.0000, A 0.000, B 0.000, C 0.000 }
gfCNCPoint2[19733] = {X 391.9492, Y 59.8676, Z -3.0000, A 0.000, B 0.000, C 0.000 }
gfCNCPoint2[19734] = {X 391.6388, Y 60.7200, Z -3.0000, A 0.000, B 0.000, C 0.000 }
gfCNCPoint2[19735] = {X 391.1157, Y 61.5158, Z -3.0000, A 0.000, B 0.000, C 0.000 }
gfCNCPoint2[19736] = {X 390.4202, Y 62.1663, Z -3.0000, A 0.000, B 0.000, C 0.000 }
gfCNCPoint2[19737] = {X 389.5912, Y 62.6349, Z -3.0000, A 0.000, B 0.000, C 0.000 }
gfCNCPoint2[19738] = {X 388.6752, Y 62.8955, Z -3.0000, A 0.000, B 0.000, C 0.000 }
gfCNCPoint2[19739] = {X 388.5090, Y 62.9185, Z -3.0000, A 0.000, B 0.000, C 0.000 }
gfCNCPoint2[19740] = {X 388.3420, Y 62.9346, Z -3.0000, A 0.000, B 0.000, C 0.000 }
gfCNCPoint2[19741] = {X 388.3383, Y 63.1540, Z -3.0000, A 0.000, B 0.000, C 0.000 }
gfCNCPoint2[19742] = {X 388.3383, Y 83.9236, Z -3.0000, A 0.000, B 0.000, C 0.000 }
gfCNCPoint2[19743] = {X 388.3363, Y 84.6159, Z -3.0000, A 0.000, B 0.000, C 0.000 }
gfCNCPoint2[19744] = {X 388.2776, Y 86.2468, Z -3.0000, A 0.000, B 0.000, C 0.000 }
gfCNCPoint2[19745] = {X 388.0766, Y 87.8663, Z -3.0000, A 0.000, B 0.000, C 0.000 }
gfCNCPoint2[19746] = {X 387.7351, Y 89.4621, Z -3.0000, A 0.000, B 0.000, C 0.000 }
gfCNCPoint2[19747] = {X 387.2173, Y 91.0069, Z -3.0000, A 0.000, B 0.000, C 0.000 }
gfCNCPoint2[19748] = {X 386.4879, Y 92.4637, Z -3.0000, A 0.000, B 0.000, C 0.000 }
gfCNCPoint2[19749] = {X 385.5613, Y 93.8038, Z -3.0000, A 0.000, B 0.000, C 0.000 }
gfCNCPoint2[19750] = {X 384.4559, Y 95.0007, Z -3.0000, A 0.000, B 0.000, C 0.000 }
gfCNCPoint2[19751] = {X 382.9677, Y 96.2544, Z -3.0000, A 0.000, B 0.000, C 0.000 }
gfCNCPoint2[19752] = {X 381.3549, Y 97.3432, Z -3.0000, A 0.000, B 0.000, C 0.000 }
gfCNCPoint2[19753] = {X 379.6357, Y 98.2546, Z -3.0000, A 0.000, B 0.000, C 0.000 }
gfCNCPoint2[19754] = {X 377.3857, Y 99.2018, Z -3.0000, A 0.000, B 0.000, C 0.000 }
gfCNCPoint2[19755] = {X 375.0734, Y 99.9847, Z -3.0000, A 0.000, B 0.000, C 0.000 }
gfCNCPoint2[19756] = {X 372.7108, Y 100.5992, Z -3.0000, A 0.000, B 0.000, C 0.000 }
gfCNCPoint2[19757] = {X 368.9146, Y 101.3336, Z -3.0000, A 0.000, B 0.000, C 0.000 }
gfCNCPoint2[19758] = {X 365.0874, Y 101.8847, Z -3.0000, A 0.000, B 0.000, C 0.000 }
gfCNCPoint2[19759] = {X 361.2381, Y 102.2512, Z -3.0000, A 0.000, B 0.000, C 0.000 }
gfCNCPoint2[19760] = {X 357.2381, Y 102.4914, Z -3.0000, A 0.000, B 0.000, C 0.000 }
gfCNCPoint2[19761] = {X 353.2337, Y 102.6447, Z -3.0000, A 0.000, B 0.000, C 0.000 }
gfCNCPoint2[19762] = {X 353.3453, Y 106.7231, Z -3.0000, A 0.000, B 0.000, C 0.000 }
gfCNCPoint2[19763] = {X 353.3453, Y 106.7231, Z 0.0000, A 0.000, B 0.000, C 0.000 }
gfCNCPoint2[19764] = {X 353.3453, Y 106.7231, Z 11.0000, A 0.000, B 0.000, C 0.000 }
gfCNCPoint2[19765] = {X 411.5991, Y 79.5931, Z 11.0000, A 0.000, B 0.000, C 0.000 }
gfCNCPoint2[19766] = {X 411.5991, Y 79.5931, Z 0.0000, A 0.000, B 0.000, C 0.000 }
gfCNCPoint2[19767] = {X 411.5991, Y 79.5931, Z -3.0000, A 0.000, B 0.000, C 0.000 }
gfCNCPoint2[19768] = {X 413.7994, Y 83.0289, Z -3.0000, A 0.000, B 0.000, C 0.000 }
gfCNCPoint2[19769] = {X 428.0552, Y 73.8994, Z -3.0000, A 0.000, B 0.000, C 0.000 }
gfCNCPoint2[19770] = {X 403.7554, Y 64.3652, Z -3.0000, A 0.000, B 0.000, C 0.000 }
gfCNCPoint2[19771] = {X 402.0596, Y 63.8036, Z -3.0000, A 0.000, B 0.000, C 0.000 }
gfCNCPoint2[19772] = {X 400.3124, Y 63.4317, Z -3.0000, A 0.000, B 0.000, C 0.000 }
gfCNCPoint2[19773] = {X 398.5349, Y 63.2540, Z -3.0000, A 0.000, B 0.000, C 0.000 }
gfCNCPoint2[19774] = {X 397.5823, Y 63.1425, Z -3.0000, A 0.000, B 0.000, C 0.000 }
gfCNCPoint2[19775] = {X 396.6779, Y 62.8236, Z -3.0000, A 0.000, B 0.000, C 0.000 }
gfCNCPoint2[19776] = {X 395.8661, Y 62.3130, Z -3.0000, A 0.000, B 0.000, C 0.000 }
gfCNCPoint2[19777] = {X 395.1869, Y 61.6359, Z -3.0000, A 0.000, B 0.000, C 0.000 }
gfCNCPoint2[19778] = {X 394.6739, Y 60.8256, Z -3.0000, A 0.000, B 0.000, C 0.000 }
gfCNCPoint2[19779] = {X 394.3522, Y 59.9221, Z -3.0000, A 0.000, B 0.000, C 0.000 }
gfCNCPoint2[19780] = {X 394.2379, Y 58.9699, Z -3.0000, A 0.000, B 0.000, C 0.000 }
gfCNCPoint2[19781] = {X 394.2377, Y 58.0000, Z -3.0000, A 0.000, B 0.000, C 0.000 }
gfCNCPoint2[19782] = {X 394.3460, Y 57.0387, Z -3.0000, A 0.000, B 0.000, C 0.000 }
gfCNCPoint2[19783] = {X 394.6655, Y 56.1256, Z -3.0000, A 0.000, B 0.000, C 0.000 }
gfCNCPoint2[19784] = {X 395.1802, Y 55.3065, Z -3.0000, A 0.000, B 0.000, C 0.000 }
gfCNCPoint2[19785] = {X 395.8642, Y 54.6225, Z -3.0000, A 0.000, B 0.000, C 0.000 }
gfCNCPoint2[19786] = {X 396.6833, Y 54.1078, Z -3.0000, A 0.000, B 0.000, C 0.000 }
gfCNCPoint2[19787] = {X 397.5964, Y 53.7883, Z -3.0000, A 0.000, B 0.000, C 0.000 }
gfCNCPoint2[19788] = {X 398.5577, Y 53.6800, Z -3.0000, A 0.000, B 0.000, C 0.000 }
gfCNCPoint2[19789] = {X 419.4886, Y 53.6800, Z -3.0000, A 0.000, B 0.000, C 0.000 }
gfCNCPoint2[19790] = {X 420.4499, Y 53.7883, Z -3.0000, A 0.000, B 0.000, C 0.000 }
gfCNCPoint2[19791] = {X 421.3630, Y 54.1078, Z -3.0000, A 0.000, B 0.000, C 0.000 }
gfCNCPoint2[19792] = {X 422.1821, Y 54.6225, Z -3.0000, A 0.000, B 0.000, C 0.000 }
gfCNCPoint2[19793] = {X 422.8661, Y 55.3065, Z -3.0000, A 0.000, B 0.000, C 0.000 }
gfCNCPoint2[19794] = {X 423.3808, Y 56.1256, Z -3.0000, A 0.000, B 0.000, C 0.000 }
gfCNCPoint2[19795] = {X 423.7003, Y 57.0387, Z -3.0000, A 0.000, B 0.000, C 0.000 }
gfCNCPoint2[19796] = {X 423.8086, Y 58.0000, Z -3.0000, A 0.000, B 0.000, C 0.000 }
gfCNCPoint2[19797] = {X 423.8086, Y 58.2325, Z -3.0000, A 0.000, B 0.000, C 0.000 }
gfCNCPoint2[19798] = {X 429.6116, Y 60.4940, Z -3.0000, A 0.000, B 0.000, C 0.000 }
gfCNCPoint2[19799] = {X 457.8608, Y 71.7019, Z -3.0000, A 0.000, B 0.000, C 0.000 }
gfCNCPoint2[19800] = {X 457.8611, Y 63.2124, Z -3.0000, A 0.000, B 0.000, C 0.000 }
gfCNCPoint2[19801] = {X 457.0093, Y 63.0034, Z -3.0000, A 0.000, B 0.000, C 0.000 }
gfCNCPoint2[19802] = {X 456.2174, Y 62.6266, Z -3.0000, A 0.000, B 0.000, C 0.000 }
gfCNCPoint2[19803] = {X 455.5178, Y 62.0977, Z -3.0000, A 0.000, B 0.000, C 0.000 }
gfCNCPoint2[19804] = {X 454.9395, Y 61.4383, Z -3.0000, A 0.000, B 0.000, C 0.000 }
gfCNCPoint2[19805] = {X 454.5063, Y 60.6758, Z -3.0000, A 0.000, B 0.000, C 0.000 }
gfCNCPoint2[19806] = {X 454.2360, Y 59.8415, Z -3.0000, A 0.000, B 0.000, C 0.000 }
gfCNCPoint2[19807] = {X 454.1398, Y 58.9697, Z -3.0000, A 0.000, B 0.000, C 0.000 }
gfCNCPoint2[19808] = {X 454.1396, Y 58.0000, Z -3.0000, A 0.000, B 0.000, C 0.000 }
gfCNCPoint2[19809] = {X 454.2479, Y 57.0387, Z -3.0000, A 0.000, B 0.000, C 0.000 }
gfCNCPoint2[19810] = {X 454.5674, Y 56.1256, Z -3.0000, A 0.000, B 0.000, C 0.000 }
gfCNCPoint2[19811] = {X 455.0821, Y 55.3065, Z -3.0000, A 0.000, B 0.000, C 0.000 }
gfCNCPoint2[19812] = {X 455.7661, Y 54.6225, Z -3.0000, A 0.000, B 0.000, C 0.000 }
gfCNCPoint2[19813] = {X 456.5852, Y 54.1078, Z -3.0000, A 0.000, B 0.000, C 0.000 }
gfCNCPoint2[19814] = {X 457.4983, Y 53.7883, Z -3.0000, A 0.000, B 0.000, C 0.000 }
gfCNCPoint2[19815] = {X 458.4596, Y 53.6800, Z -3.0000, A 0.000, B 0.000, C 0.000 }
gfCNCPoint2[19816] = {X 475.0000, Y 53.6800, Z -3.0000, A 0.000, B 0.000, C 0.000 }
gfCNCPoint2[19817] = {X 475.9613, Y 53.7883, Z -3.0000, A 0.000, B 0.000, C 0.000 }
gfCNCPoint2[19818] = {X 476.8744, Y 54.1078, Z -3.0000, A 0.000, B 0.000, C 0.000 }
gfCNCPoint2[19819] = {X 477.6935, Y 54.6225, Z -3.0000, A 0.000, B 0.000, C 0.000 }
gfCNCPoint2[19820] = {X 478.3775, Y 55.3065, Z -3.0000, A 0.000, B 0.000, C 0.000 }
gfCNCPoint2[19821] = {X 478.8922, Y 56.1256, Z -3.0000, A 0.000, B 0.000, C 0.000 }
gfCNCPoint2[19822] = {X 479.2117, Y 57.0387, Z -3.0000, A 0.000, B 0.000, C 0.000 }
gfCNCPoint2[19823] = {X 479.3200, Y 58.0000, Z -3.0000, A 0.000, B 0.000, C 0.000 }
gfCNCPoint2[19824] = {X 479.3200, Y 58.9342, Z -3.0000, A 0.000, B 0.000, C 0.000 }
gfCNCPoint2[19825] = {X 479.2300, Y 59.8115, Z -3.0000, A 0.000, B 0.000, C 0.000 }
gfCNCPoint2[19826] = {X 478.9636, Y 60.6522, Z -3.0000, A 0.000, B 0.000, C 0.000 }
gfCNCPoint2[19827] = {X 478.5321, Y 61.4213, Z -3.0000, A 0.000, B 0.000, C 0.000 }
gfCNCPoint2[19828] = {X 477.9534, Y 62.0868, Z -3.0000, A 0.000, B 0.000, C 0.000 }
gfCNCPoint2[19829] = {X 477.2516, Y 62.6209, Z -3.0000, A 0.000, B 0.000, C 0.000 }
gfCNCPoint2[19830] = {X 476.4560, Y 63.0013, Z -3.0000, A 0.000, B 0.000, C 0.000 }
gfCNCPoint2[19831] = {X 475.5997, Y 63.2122, Z -3.0000, A 0.000, B 0.000, C 0.000 }
gfCNCPoint2[19832] = {X 475.6001, Y 92.7686, Z -3.0000, A 0.000, B 0.000, C 0.000 }
gfCNCPoint2[19833] = {X 475.9962, Y 92.8676, Z -3.0000, A 0.000, B 0.000, C 0.000 }
gfCNCPoint2[19834] = {X 476.3866, Y 92.9870, Z -3.0000, A 0.000, B 0.000, C 0.000 }
gfCNCPoint2[19835] = {X 477.1986, Y 93.3558, Z -3.0000, A 0.000, B 0.000, C 0.000 }
gfCNCPoint2[19836] = {X 477.9168, Y 93.8845, Z -3.0000, A 0.000, B 0.000, C 0.000 }
gfCNCPoint2[19837] = {X 478.5103, Y 94.5500, Z -3.0000, A 0.000, B 0.000, C 0.000 }
gfCNCPoint2[19838] = {X 478.9536, Y 95.3239, Z -3.0000, A 0.000, B 0.000, C 0.000 }
gfCNCPoint2[19839] = {X 479.2274, Y 96.1726, Z -3.0000, A 0.000, B 0.000, C 0.000 }
gfCNCPoint2[19840] = {X 479.3200, Y 97.0595, Z -3.0000, A 0.000, B 0.000, C 0.000 }
gfCNCPoint2[19841] = {X 479.3200, Y 98.0000, Z -3.0000, A 0.000, B 0.000, C 0.000 }
gfCNCPoint2[19842] = {X 479.2117, Y 98.9613, Z -3.0000, A 0.000, B 0.000, C 0.000 }
gfCNCPoint2[19843] = {X 478.8922, Y 99.8744, Z -3.0000, A 0.000, B 0.000, C 0.000 }
gfCNCPoint2[19844] = {X 478.3775, Y 100.6935, Z -3.0000, A 0.000, B 0.000, C 0.000 }
gfCNCPoint2[19845] = {X 477.6935, Y 101.3775, Z -3.0000, A 0.000, B 0.000, C 0.000 }
gfCNCPoint2[19846] = {X 476.8744, Y 101.8922, Z -3.0000, A 0.000, B 0.000, C 0.000 }
gfCNCPoint2[19847] = {X 475.9613, Y 102.2117, Z -3.0000, A 0.000, B 0.000, C 0.000 }
gfCNCPoint2[19848] = {X 475.0000, Y 102.3200, Z -3.0000, A 0.000, B 0.000, C 0.000 }
gfCNCPoint2[19849] = {X 458.4596, Y 102.3200, Z -3.0000, A 0.000, B 0.000, C 0.000 }
gfCNCPoint2[19850] = {X 457.4983, Y 102.2117, Z -3.0000, A 0.000, B 0.000, C 0.000 }
gfCNCPoint2[19851] = {X 456.5852, Y 101.8922, Z -3.0000, A 0.000, B 0.000, C 0.000 }
gfCNCPoint2[19852] = {X 455.7661, Y 101.3775, Z -3.0000, A 0.000, B 0.000, C 0.000 }
gfCNCPoint2[19853] = {X 455.0821, Y 100.6935, Z -3.0000, A 0.000, B 0.000, C 0.000 }
gfCNCPoint2[19854] = {X 454.5674, Y 99.8744, Z -3.0000, A 0.000, B 0.000, C 0.000 }
gfCNCPoint2[19855] = {X 454.2479, Y 98.9613, Z -3.0000, A 0.000, B 0.000, C 0.000 }
gfCNCPoint2[19856] = {X 454.1396, Y 98.0000, Z -3.0000, A 0.000, B 0.000, C 0.000 }
gfCNCPoint2[19857] = {X 454.1396, Y 97.0659, Z -3.0000, A 0.000, B 0.000, C 0.000 }
gfCNCPoint2[19858] = {X 454.2295, Y 96.1891, Z -3.0000, A 0.000, B 0.000, C 0.000 }
gfCNCPoint2[19859] = {X 454.4955, Y 95.3488, Z -3.0000, A 0.000, B 0.000, C 0.000 }
gfCNCPoint2[19860] = {X 454.9265, Y 94.5800, Z -3.0000, A 0.000, B 0.000, C 0.000 }
gfCNCPoint2[19861] = {X 455.5046, Y 93.9147, Z -3.0000, A 0.000, B 0.000, C 0.000 }
gfCNCPoint2[19862] = {X 456.2057, Y 93.3805, Z -3.0000, A 0.000, B 0.000, C 0.000 }
gfCNCPoint2[19863] = {X 457.0006, Y 92.9998, Z -3.0000, A 0.000, B 0.000, C 0.000 }
gfCNCPoint2[19864] = {X 457.8563, Y 92.7883, Z -3.0000, A 0.000, B 0.000, C 0.000 }
gfCNCPoint2[19865] = {X 457.8563, Y 85.5950, Z -3.0000, A 0.000, B 0.000, C 0.000 }
gfCNCPoint2[19866] = {X 444.8585, Y 80.4998, Z -3.0000, A 0.000, B 0.000, C 0.000 }
gfCNCPoint2[19867] = {X 420.0230, Y 96.5881, Z -3.0000, A 0.000, B 0.000, C 0.000 }
gfCNCPoint2[19868] = {X 420.0267, Y 97.0647, Z -3.0000, A 0.000, B 0.000, C 0.000 }
gfCNCPoint2[19869] = {X 420.0267, Y 98.0000, Z -3.0000, A 0.000, B 0.000, C 0.000 }
gfCNCPoint2[19870] = {X 419.9184, Y 98.9613, Z -3.0000, A 0.000, B 0.000, C 0.000 }
gfCNCPoint2[19871] = {X 419.5989, Y 99.8744, Z -3.0000, A 0.000, B 0.000, C 0.000 }
gfCNCPoint2[19872] = {X 419.0842, Y 100.6935, Z -3.0000, A 0.000, B 0.000, C 0.000 }
gfCNCPoint2[19873] = {X 418.4002, Y 101.3775, Z -3.0000, A 0.000, B 0.000, C 0.000 }
gfCNCPoint2[19874] = {X 417.5811, Y 101.8922, Z -3.0000, A 0.000, B 0.000, C 0.000 }
gfCNCPoint2[19875] = {X 416.6680, Y 102.2117, Z -3.0000, A 0.000, B 0.000, C 0.000 }
gfCNCPoint2[19876] = {X 415.7067, Y 102.3200, Z -3.0000, A 0.000, B 0.000, C 0.000 }
gfCNCPoint2[19877] = {X 396.4059, Y 102.3200, Z -3.0000, A 0.000, B 0.000, C 0.000 }
gfCNCPoint2[19878] = {X 395.4447, Y 102.2117, Z -3.0000, A 0.000, B 0.000, C 0.000 }
gfCNCPoint2[19879] = {X 394.5316, Y 101.8922, Z -3.0000, A 0.000, B 0.000, C 0.000 }
gfCNCPoint2[19880] = {X 393.7125, Y 101.3775, Z -3.0000, A 0.000, B 0.000, C 0.000 }
gfCNCPoint2[19881] = {X 393.0284, Y 100.6935, Z -3.0000, A 0.000, B 0.000, C 0.000 }
gfCNCPoint2[19882] = {X 392.5138, Y 99.8744, Z -3.0000, A 0.000, B 0.000, C 0.000 }
gfCNCPoint2[19883] = {X 392.1943, Y 98.9613, Z -3.0000, A 0.000, B 0.000, C 0.000 }
gfCNCPoint2[19884] = {X 392.0859, Y 98.0000, Z -3.0000, A 0.000, B 0.000, C 0.000 }
gfCNCPoint2[19885] = {X 392.0859, Y 97.0659, Z -3.0000, A 0.000, B 0.000, C 0.000 }
gfCNCPoint2[19886] = {X 392.1938, Y 96.1069, Z -3.0000, A 0.000, B 0.000, C 0.000 }
gfCNCPoint2[19887] = {X 392.5118, Y 95.1957, Z -3.0000, A 0.000, B 0.000, C 0.000 }
gfCNCPoint2[19888] = {X 393.0242, Y 94.3778, Z -3.0000, A 0.000, B 0.000, C 0.000 }
gfCNCPoint2[19889] = {X 393.7054, Y 93.6941, Z -3.0000, A 0.000, B 0.000, C 0.000 }
gfCNCPoint2[19890] = {X 394.5213, Y 93.1787, Z -3.0000, A 0.000, B 0.000, C 0.000 }
gfCNCPoint2[19891] = {X 395.4314, Y 92.8573, Z -3.0000, A 0.000, B 0.000, C 0.000 }
gfCNCPoint2[19892] = {X 396.3900, Y 92.7460, Z -3.0000, A 0.000, B 0.000, C 0.000 }
gfCNCPoint2[19893] = {X 397.3434, Y 92.7053, Z -3.0000, A 0.000, B 0.000, C 0.000 }
gfCNCPoint2[19894] = {X 398.2933, Y 92.6150, Z -3.0000, A 0.000, B 0.000, C 0.000 }
gfCNCPoint2[19895] = {X 398.9443, Y 92.4573, Z -3.0000, A 0.000, B 0.000, C 0.000 }
gfCNCPoint2[19896] = {X 399.5436, Y 92.1583, Z -3.0000, A 0.000, B 0.000, C 0.000 }
gfCNCPoint2[19897] = {X 413.7994, Y 83.0289, Z -3.0000, A 0.000, B 0.000, C 0.000 }
gfCNCPoint2[19898] = {X 411.6422, Y 79.6604, Z -3.0000, A 0.000, B 0.000, C 0.000 }
gfCNCPoint2[19899] = {X 413.8425, Y 83.0963, Z -3.0000, A 0.000, B 0.000, C 0.000 }
gfCNCPoint2[19900] = {X 428.2304, Y 73.8823, Z -3.0000, A 0.000, B 0.000, C 0.000 }
gfCNCPoint2[19901] = {X 403.7847, Y 64.2907, Z -3.0000, A 0.000, B 0.000, C 0.000 }
gfCNCPoint2[19902] = {X 402.0800, Y 63.7263, Z -3.0000, A 0.000, B 0.000, C 0.000 }
gfCNCPoint2[19903] = {X 400.3237, Y 63.3525, Z -3.0000, A 0.000, B 0.000, C 0.000 }
gfCNCPoint2[19904] = {X 398.5369, Y 63.1740, Z -3.0000, A 0.000, B 0.000, C 0.000 }
gfCNCPoint2[19905] = {X 397.6017, Y 63.0649, Z -3.0000, A 0.000, B 0.000, C 0.000 }
gfCNCPoint2[19906] = {X 396.7137, Y 62.7521, Z -3.0000, A 0.000, B 0.000, C 0.000 }
gfCNCPoint2[19907] = {X 395.9166, Y 62.2510, Z -3.0000, A 0.000, B 0.000, C 0.000 }
gfCNCPoint2[19908] = {X 395.2497, Y 61.5864, Z -3.0000, A 0.000, B 0.000, C 0.000 }
gfCNCPoint2[19909] = {X 394.7460, Y 60.7910, Z -3.0000, A 0.000, B 0.000, C 0.000 }
gfCNCPoint2[19910] = {X 394.4302, Y 59.9041, Z -3.0000, A 0.000, B 0.000, C 0.000 }
gfCNCPoint2[19911] = {X 394.3179, Y 58.9693, Z -3.0000, A 0.000, B 0.000, C 0.000 }
gfCNCPoint2[19912] = {X 394.3177, Y 58.0000, Z -3.0000, A 0.000, B 0.000, C 0.000 }
gfCNCPoint2[19913] = {X 394.4240, Y 57.0565, Z -3.0000, A 0.000, B 0.000, C 0.000 }
gfCNCPoint2[19914] = {X 394.7376, Y 56.1603, Z -3.0000, A 0.000, B 0.000, C 0.000 }
gfCNCPoint2[19915] = {X 395.2428, Y 55.3564, Z -3.0000, A 0.000, B 0.000, C 0.000 }
gfCNCPoint2[19916] = {X 395.9141, Y 54.6850, Z -3.0000, A 0.000, B 0.000, C 0.000 }
gfCNCPoint2[19917] = {X 396.7181, Y 54.1799, Z -3.0000, A 0.000, B 0.000, C 0.000 }
gfCNCPoint2[19918] = {X 397.6142, Y 53.8663, Z -3.0000, A 0.000, B 0.000, C 0.000 }
gfCNCPoint2[19919] = {X 398.5577, Y 53.7600, Z -3.0000, A 0.000, B 0.000, C 0.000 }
gfCNCPoint2[19920] = {X 419.4886, Y 53.7600, Z -3.0000, A 0.000, B 0.000, C 0.000 }
gfCNCPoint2[19921] = {X 420.4321, Y 53.8663, Z -3.0000, A 0.000, B 0.000, C 0.000 }
gfCNCPoint2[19922] = {X 421.3283, Y 54.1799, Z -3.0000, A 0.000, B 0.000, C 0.000 }
gfCNCPoint2[19923] = {X 422.1322, Y 54.6850, Z -3.0000, A 0.000, B 0.000, C 0.000 }
gfCNCPoint2[19924] = {X 422.8036, Y 55.3564, Z -3.0000, A 0.000, B 0.000, C 0.000 }
gfCNCPoint2[19925] = {X 423.3087, Y 56.1603, Z -3.0000, A 0.000, B 0.000, C 0.000 }
gfCNCPoint2[19926] = {X 423.6223, Y 57.0565, Z -3.0000, A 0.000, B 0.000, C 0.000 }
gfCNCPoint2[19927] = {X 423.7286, Y 58.0000, Z -3.0000, A 0.000, B 0.000, C 0.000 }
gfCNCPoint2[19928] = {X 423.7286, Y 58.2872, Z -3.0000, A 0.000, B 0.000, C 0.000 }
gfCNCPoint2[19929] = {X 429.5823, Y 60.5685, Z -3.0000, A 0.000, B 0.000, C 0.000 }
gfCNCPoint2[19930] = {X 457.9408, Y 71.8197, Z -3.0000, A 0.000, B 0.000, C 0.000 }
gfCNCPoint2[19931] = {X 457.9411, Y 63.1422, Z -3.0000, A 0.000, B 0.000, C 0.000 }
gfCNCPoint2[19932] = {X 457.0925, Y 62.9476, Z -3.0000, A 0.000, B 0.000, C 0.000 }
gfCNCPoint2[19933] = {X 456.3015, Y 62.5837, Z -3.0000, A 0.000, B 0.000, C 0.000 }
gfCNCPoint2[19934] = {X 455.6015, Y 62.0660, Z -3.0000, A 0.000, B 0.000, C 0.000 }
gfCNCPoint2[19935] = {X 455.0220, Y 61.4162, Z -3.0000, A 0.000, B 0.000, C 0.000 }
gfCNCPoint2[19936] = {X 454.5875, Y 60.6617, Z -3.0000, A 0.000, B 0.000, C 0.000 }
gfCNCPoint2[19937] = {X 454.3163, Y 59.8344, Z -3.0000, A 0.000, B 0.000, C 0.000 }
gfCNCPoint2[19938] = {X 454.2197, Y 58.9691, Z -3.0000, A 0.000, B 0.000, C 0.000 }
gfCNCPoint2[19939] = {X 454.2196, Y 58.0000, Z -3.0000, A 0.000, B 0.000, C 0.000 }
gfCNCPoint2[19940] = {X 454.3259, Y 57.0565, Z -3.0000, A 0.000, B 0.000, C 0.000 }
gfCNCPoint2[19941] = {X 454.6395, Y 56.1603, Z -3.0000, A 0.000, B 0.000, C 0.000 }
gfCNCPoint2[19942] = {X 455.1446, Y 55.3564, Z -3.0000, A 0.000, B 0.000, C 0.000 }
gfCNCPoint2[19943] = {X 455.8160, Y 54.6850, Z -3.0000, A 0.000, B 0.000, C 0.000 }
gfCNCPoint2[19944] = {X 456.6199, Y 54.1799, Z -3.0000, A 0.000, B 0.000, C 0.000 }
gfCNCPoint2[19945] = {X 457.5161, Y 53.8663, Z -3.0000, A 0.000, B 0.000, C 0.000 }
gfCNCPoint2[19946] = {X 458.4596, Y 53.7600, Z -3.0000, A 0.000, B 0.000, C 0.000 }
gfCNCPoint2[19947] = {X 475.0000, Y 53.7600, Z -3.0000, A 0.000, B 0.000, C 0.000 }
gfCNCPoint2[19948] = {X 475.9435, Y 53.8663, Z -3.0000, A 0.000, B 0.000, C 0.000 }
gfCNCPoint2[19949] = {X 476.8397, Y 54.1799, Z -3.0000, A 0.000, B 0.000, C 0.000 }
gfCNCPoint2[19950] = {X 477.6436, Y 54.6850, Z -3.0000, A 0.000, B 0.000, C 0.000 }
gfCNCPoint2[19951] = {X 478.3150, Y 55.3564, Z -3.0000, A 0.000, B 0.000, C 0.000 }
gfCNCPoint2[19952] = {X 478.8201, Y 56.1603, Z -3.0000, A 0.000, B 0.000, C 0.000 }
gfCNCPoint2[19953] = {X 479.1337, Y 57.0565, Z -3.0000, A 0.000, B 0.000, C 0.000 }
gfCNCPoint2[19954] = {X 479.2400, Y 58.0000, Z -3.0000, A 0.000, B 0.000, C 0.000 }
gfCNCPoint2[19955] = {X 479.2400, Y 58.9342, Z -3.0000, A 0.000, B 0.000, C 0.000 }
gfCNCPoint2[19956] = {X 479.1496, Y 59.8050, Z -3.0000, A 0.000, B 0.000, C 0.000 }
gfCNCPoint2[19957] = {X 478.8823, Y 60.6386, Z -3.0000, A 0.000, B 0.000, C 0.000 }
gfCNCPoint2[19958] = {X 478.4495, Y 61.3996, Z -3.0000, A 0.000, B 0.000, C 0.000 }
gfCNCPoint2[19959] = {X 477.8696, Y 62.0554, Z -3.0000, A 0.000, B 0.000, C 0.000 }
gfCNCPoint2[19960] = {X 477.1674, Y 62.5782, Z -3.0000, A 0.000, B 0.000, C 0.000 }
gfCNCPoint2[19961] = {X 476.3728, Y 62.9457, Z -3.0000, A 0.000, B 0.000, C 0.000 }
gfCNCPoint2[19962] = {X 475.5197, Y 63.1421, Z -3.0000, A 0.000, B 0.000, C 0.000 }
gfCNCPoint2[19963] = {X 475.5201, Y 92.8330, Z -3.0000, A 0.000, B 0.000, C 0.000 }
gfCNCPoint2[19964] = {X 475.9439, Y 92.9362, Z -3.0000, A 0.000, B 0.000, C 0.000 }
gfCNCPoint2[19965] = {X 476.3613, Y 93.0628, Z -3.0000, A 0.000, B 0.000, C 0.000 }
gfCNCPoint2[19966] = {X 477.1581, Y 93.4248, Z -3.0000, A 0.000, B 0.000, C 0.000 }
gfCNCPoint2[19967] = {X 477.8629, Y 93.9436, Z -3.0000, A 0.000, B 0.000, C 0.000 }
gfCNCPoint2[19968] = {X 478.4454, Y 94.5968, Z -3.0000, A 0.000, B 0.000, C 0.000 }
gfCNCPoint2[19969] = {X 478.8804, Y 95.3562, Z -3.0000, A 0.000, B 0.000, C 0.000 }
gfCNCPoint2[19970] = {X 479.1491, Y 96.1891, Z -3.0000, A 0.000, B 0.000, C 0.000 }
gfCNCPoint2[19971] = {X 479.2400, Y 97.0595, Z -3.0000, A 0.000, B 0.000, C 0.000 }
gfCNCPoint2[19972] = {X 479.2400, Y 98.0000, Z -3.0000, A 0.000, B 0.000, C 0.000 }
gfCNCPoint2[19973] = {X 479.1337, Y 98.9435, Z -3.0000, A 0.000, B 0.000, C 0.000 }
gfCNCPoint2[19974] = {X 478.8201, Y 99.8397, Z -3.0000, A 0.000, B 0.000, C 0.000 }
gfCNCPoint2[19975] = {X 478.3150, Y 100.6436, Z -3.0000, A 0.000, B 0.000, C 0.000 }
gfCNCPoint2[19976] = {X 477.6436, Y 101.3150, Z -3.0000, A 0.000, B 0.000, C 0.000 }
gfCNCPoint2[19977] = {X 476.8397, Y 101.8201, Z -3.0000, A 0.000, B 0.000, C 0.000 }
gfCNCPoint2[19978] = {X 475.9435, Y 102.1337, Z -3.0000, A 0.000, B 0.000, C 0.000 }
gfCNCPoint2[19979] = {X 475.0000, Y 102.2400, Z -3.0000, A 0.000, B 0.000, C 0.000 }
gfCNCPoint2[19980] = {X 458.4596, Y 102.2400, Z -3.0000, A 0.000, B 0.000, C 0.000 }
gfCNCPoint2[19981] = {X 457.5161, Y 102.1337, Z -3.0000, A 0.000, B 0.000, C 0.000 }
gfCNCPoint2[19982] = {X 456.6199, Y 101.8201, Z -3.0000, A 0.000, B 0.000, C 0.000 }
gfCNCPoint2[19983] = {X 455.8160, Y 101.3150, Z -3.0000, A 0.000, B 0.000, C 0.000 }
gfCNCPoint2[19984] = {X 455.1446, Y 100.6436, Z -3.0000, A 0.000, B 0.000, C 0.000 }
gfCNCPoint2[19985] = {X 454.6395, Y 99.8397, Z -3.0000, A 0.000, B 0.000, C 0.000 }
gfCNCPoint2[19986] = {X 454.3259, Y 98.9435, Z -3.0000, A 0.000, B 0.000, C 0.000 }
gfCNCPoint2[19987] = {X 454.2196, Y 98.0000, Z -3.0000, A 0.000, B 0.000, C 0.000 }
gfCNCPoint2[19988] = {X 454.2196, Y 97.0659, Z -3.0000, A 0.000, B 0.000, C 0.000 }
gfCNCPoint2[19989] = {X 454.3099, Y 96.1957, Z -3.0000, A 0.000, B 0.000, C 0.000 }
gfCNCPoint2[19990] = {X 454.5769, Y 95.3624, Z -3.0000, A 0.000, B 0.000, C 0.000 }
gfCNCPoint2[19991] = {X 455.0092, Y 94.6018, Z -3.0000, A 0.000, B 0.000, C 0.000 }
gfCNCPoint2[19992] = {X 455.5884, Y 93.9460, Z -3.0000, A 0.000, B 0.000, C 0.000 }
gfCNCPoint2[19993] = {X 456.2899, Y 93.4231, Z -3.0000, A 0.000, B 0.000, C 0.000 }
gfCNCPoint2[19994] = {X 457.0838, Y 93.0553, Z -3.0000, A 0.000, B 0.000, C 0.000 }
gfCNCPoint2[19995] = {X 457.9363, Y 92.8584, Z -3.0000, A 0.000, B 0.000, C 0.000 }
gfCNCPoint2[19996] = {X 457.9363, Y 85.5404, Z -3.0000, A 0.000, B 0.000, C 0.000 }
gfCNCPoint2[19997] = {X 444.8494, Y 80.4103, Z -3.0000, A 0.000, B 0.000, C 0.000 }
gfCNCPoint2[19998] = {X 419.9426, Y 96.5448, Z -3.0000, A 0.000, B 0.000, C 0.000 }
gfCNCPoint2[19999] = {X 419.9467, Y 97.0650, Z -3.0000, A 0.000, B 0.000, C 0.000 }
gfCNCPoint2[20000] = {X 419.9467, Y 98.0000, Z -3.0000, A 0.000, B 0.000, C 0.000 }
gfCNCPoint2[20001] = {X 419.8404, Y 98.9435, Z -3.0000, A 0.000, B 0.000, C 0.000 }
gfCNCPoint2[20002] = {X 419.5268, Y 99.8397, Z -3.0000, A 0.000, B 0.000, C 0.000 }
gfCNCPoint2[20003] = {X 419.0217, Y 100.6436, Z -3.0000, A 0.000, B 0.000, C 0.000 }
gfCNCPoint2[20004] = {X 418.3503, Y 101.3150, Z -3.0000, A 0.000, B 0.000, C 0.000 }
gfCNCPoint2[20005] = {X 417.5464, Y 101.8201, Z -3.0000, A 0.000, B 0.000, C 0.000 }
gfCNCPoint2[20006] = {X 416.6502, Y 102.1337, Z -3.0000, A 0.000, B 0.000, C 0.000 }
gfCNCPoint2[20007] = {X 415.7067, Y 102.2400, Z -3.0000, A 0.000, B 0.000, C 0.000 }
gfCNCPoint2[20008] = {X 396.4059, Y 102.2400, Z -3.0000, A 0.000, B 0.000, C 0.000 }
gfCNCPoint2[20009] = {X 395.4625, Y 102.1337, Z -3.0000, A 0.000, B 0.000, C 0.000 }
gfCNCPoint2[20010] = {X 394.5663, Y 101.8201, Z -3.0000, A 0.000, B 0.000, C 0.000 }
gfCNCPoint2[20011] = {X 393.7624, Y 101.3150, Z -3.0000, A 0.000, B 0.000, C 0.000 }
gfCNCPoint2[20012] = {X 393.0910, Y 100.6436, Z -3.0000, A 0.000, B 0.000, C 0.000 }
gfCNCPoint2[20013] = {X 392.5858, Y 99.8397, Z -3.0000, A 0.000, B 0.000, C 0.000 }
gfCNCPoint2[20014] = {X 392.2723, Y 98.9435, Z -3.0000, A 0.000, B 0.000, C 0.000 }
gfCNCPoint2[20015] = {X 392.1659, Y 98.0000, Z -3.0000, A 0.000, B 0.000, C 0.000 }
gfCNCPoint2[20016] = {X 392.1659, Y 97.0659, Z -3.0000, A 0.000, B 0.000, C 0.000 }
gfCNCPoint2[20017] = {X 392.2718, Y 96.1245, Z -3.0000, A 0.000, B 0.000, C 0.000 }
gfCNCPoint2[20018] = {X 392.5840, Y 95.2301, Z -3.0000, A 0.000, B 0.000, C 0.000 }
gfCNCPoint2[20019] = {X 393.0870, Y 94.4274, Z -3.0000, A 0.000, B 0.000, C 0.000 }
gfCNCPoint2[20020] = {X 393.7556, Y 93.7563, Z -3.0000, A 0.000, B 0.000, C 0.000 }
gfCNCPoint2[20021] = {X 394.5566, Y 93.2505, Z -3.0000, A 0.000, B 0.000, C 0.000 }
gfCNCPoint2[20022] = {X 395.4499, Y 92.9351, Z -3.0000, A 0.000, B 0.000, C 0.000 }
gfCNCPoint2[20023] = {X 396.3909, Y 92.8260, Z -3.0000, A 0.000, B 0.000, C 0.000 }
gfCNCPoint2[20024] = {X 397.3488, Y 92.7851, Z -3.0000, A 0.000, B 0.000, C 0.000 }
gfCNCPoint2[20025] = {X 398.3032, Y 92.6944, Z -3.0000, A 0.000, B 0.000, C 0.000 }
gfCNCPoint2[20026] = {X 398.9717, Y 92.5325, Z -3.0000, A 0.000, B 0.000, C 0.000 }
gfCNCPoint2[20027] = {X 399.5871, Y 92.2255, Z -3.0000, A 0.000, B 0.000, C 0.000 }
gfCNCPoint2[20028] = {X 413.8425, Y 83.0963, Z -3.0000, A 0.000, B 0.000, C 0.000 }
gfCNCPoint2[20029] = {X 411.6854, Y 79.7278, Z -3.0000, A 0.000, B 0.000, C 0.000 }
gfCNCPoint2[20030] = {X 413.8857, Y 83.1636, Z -3.0000, A 0.000, B 0.000, C 0.000 }
gfCNCPoint2[20031] = {X 428.4056, Y 73.8651, Z -3.0000, A 0.000, B 0.000, C 0.000 }
gfCNCPoint2[20032] = {X 403.8140, Y 64.2163, Z -3.0000, A 0.000, B 0.000, C 0.000 }
gfCNCPoint2[20033] = {X 402.1005, Y 63.6489, Z -3.0000, A 0.000, B 0.000, C 0.000 }
gfCNCPoint2[20034] = {X 400.3349, Y 63.2733, Z -3.0000, A 0.000, B 0.000, C 0.000 }
gfCNCPoint2[20035] = {X 398.5388, Y 63.0940, Z -3.0000, A 0.000, B 0.000, C 0.000 }
gfCNCPoint2[20036] = {X 397.6211, Y 62.9872, Z -3.0000, A 0.000, B 0.000, C 0.000 }
gfCNCPoint2[20037] = {X 396.7495, Y 62.6805, Z -3.0000, A 0.000, B 0.000, C 0.000 }
gfCNCPoint2[20038] = {X 395.9671, Y 62.1890, Z -3.0000, A 0.000, B 0.000, C 0.000 }
gfCNCPoint2[20039] = {X 395.3126, Y 61.5369, Z -3.0000, A 0.000, B 0.000, C 0.000 }
gfCNCPoint2[20040] = {X 394.8181, Y 60.7564, Z -3.0000, A 0.000, B 0.000, C 0.000 }
gfCNCPoint2[20041] = {X 394.5081, Y 59.8860, Z -3.0000, A 0.000, B 0.000, C 0.000 }
gfCNCPoint2[20042] = {X 394.3979, Y 58.9686, Z -3.0000, A 0.000, B 0.000, C 0.000 }
gfCNCPoint2[20043] = {X 394.3977, Y 58.0000, Z -3.0000, A 0.000, B 0.000, C 0.000 }
gfCNCPoint2[20044] = {X 394.5020, Y 57.0743, Z -3.0000, A 0.000, B 0.000, C 0.000 }
gfCNCPoint2[20045] = {X 394.8097, Y 56.1950, Z -3.0000, A 0.000, B 0.000, C 0.000 }
gfCNCPoint2[20046] = {X 395.3053, Y 55.4063, Z -3.0000, A 0.000, B 0.000, C 0.000 }
gfCNCPoint2[20047] = {X 395.9640, Y 54.7476, Z -3.0000, A 0.000, B 0.000, C 0.000 }
gfCNCPoint2[20048] = {X 396.7528, Y 54.2520, Z -3.0000, A 0.000, B 0.000, C 0.000 }
gfCNCPoint2[20049] = {X 397.6320, Y 53.9443, Z -3.0000, A 0.000, B 0.000, C 0.000 }
gfCNCPoint2[20050] = {X 398.5577, Y 53.8400, Z -3.0000, A 0.000, B 0.000, C 0.000 }
gfCNCPoint2[20051] = {X 419.4886, Y 53.8400, Z -3.0000, A 0.000, B 0.000, C 0.000 }
gfCNCPoint2[20052] = {X 420.4143, Y 53.9443, Z -3.0000, A 0.000, B 0.000, C 0.000 }
gfCNCPoint2[20053] = {X 421.2936, Y 54.2520, Z -3.0000, A 0.000, B 0.000, C 0.000 }
gfCNCPoint2[20054] = {X 422.0823, Y 54.7476, Z -3.0000, A 0.000, B 0.000, C 0.000 }
gfCNCPoint2[20055] = {X 422.7410, Y 55.4063, Z -3.0000, A 0.000, B 0.000, C 0.000 }
gfCNCPoint2[20056] = {X 423.2366, Y 56.1950, Z -3.0000, A 0.000, B 0.000, C 0.000 }
gfCNCPoint2[20057] = {X 423.5443, Y 57.0743, Z -3.0000, A 0.000, B 0.000, C 0.000 }
gfCNCPoint2[20058] = {X 423.6486, Y 58.0000, Z -3.0000, A 0.000, B 0.000, C 0.000 }
gfCNCPoint2[20059] = {X 423.6486, Y 58.3419, Z -3.0000, A 0.000, B 0.000, C 0.000 }
gfCNCPoint2[20060] = {X 429.5531, Y 60.6429, Z -3.0000, A 0.000, B 0.000, C 0.000 }
gfCNCPoint2[20061] = {X 458.0208, Y 71.9375, Z -3.0000, A 0.000, B 0.000, C 0.000 }
gfCNCPoint2[20062] = {X 458.0211, Y 63.0709, Z -3.0000, A 0.000, B 0.000, C 0.000 }
gfCNCPoint2[20063] = {X 457.9187, Y 63.0588, Z -3.0000, A 0.000, B 0.000, C 0.000 }
gfCNCPoint2[20064] = {X 457.8167, Y 63.0441, Z -3.0000, A 0.000, B 0.000, C 0.000 }
gfCNCPoint2[20065] = {X 456.8790, Y 62.7821, Z -3.0000, A 0.000, B 0.000, C 0.000 }
gfCNCPoint2[20066] = {X 456.0280, Y 62.3094, Z -3.0000, A 0.000, B 0.000, C 0.000 }
gfCNCPoint2[20067] = {X 455.3101, Y 61.6518, Z -3.0000, A 0.000, B 0.000, C 0.000 }
gfCNCPoint2[20068] = {X 454.7647, Y 60.8454, Z -3.0000, A 0.000, B 0.000, C 0.000 }
gfCNCPoint2[20069] = {X 454.4216, Y 59.9343, Z -3.0000, A 0.000, B 0.000, C 0.000 }
gfCNCPoint2[20070] = {X 454.2997, Y 58.9684, Z -3.0000, A 0.000, B 0.000, C 0.000 }
gfCNCPoint2[20071] = {X 454.2996, Y 58.0000, Z -3.0000, A 0.000, B 0.000, C 0.000 }
gfCNCPoint2[20072] = {X 454.4039, Y 57.0743, Z -3.0000, A 0.000, B 0.000, C 0.000 }
gfCNCPoint2[20073] = {X 454.7116, Y 56.1950, Z -3.0000, A 0.000, B 0.000, C 0.000 }
gfCNCPoint2[20074] = {X 455.2072, Y 55.4063, Z -3.0000, A 0.000, B 0.000, C 0.000 }
gfCNCPoint2[20075] = {X 455.8659, Y 54.7476, Z -3.0000, A 0.000, B 0.000, C 0.000 }
gfCNCPoint2[20076] = {X 456.6546, Y 54.2520, Z -3.0000, A 0.000, B 0.000, C 0.000 }
gfCNCPoint2[20077] = {X 457.5339, Y 53.9443, Z -3.0000, A 0.000, B 0.000, C 0.000 }
gfCNCPoint2[20078] = {X 458.4596, Y 53.8400, Z -3.0000, A 0.000, B 0.000, C 0.000 }
gfCNCPoint2[20079] = {X 475.0000, Y 53.8400, Z -3.0000, A 0.000, B 0.000, C 0.000 }
gfCNCPoint2[20080] = {X 475.9257, Y 53.9443, Z -3.0000, A 0.000, B 0.000, C 0.000 }
gfCNCPoint2[20081] = {X 476.8050, Y 54.2520, Z -3.0000, A 0.000, B 0.000, C 0.000 }
gfCNCPoint2[20082] = {X 477.5937, Y 54.7476, Z -3.0000, A 0.000, B 0.000, C 0.000 }
gfCNCPoint2[20083] = {X 478.2524, Y 55.4063, Z -3.0000, A 0.000, B 0.000, C 0.000 }
gfCNCPoint2[20084] = {X 478.7480, Y 56.1950, Z -3.0000, A 0.000, B 0.000, C 0.000 }
gfCNCPoint2[20085] = {X 479.0557, Y 57.0743, Z -3.0000, A 0.000, B 0.000, C 0.000 }
gfCNCPoint2[20086] = {X 479.1600, Y 58.0000, Z -3.0000, A 0.000, B 0.000, C 0.000 }
gfCNCPoint2[20087] = {X 479.1600, Y 58.9342, Z -3.0000, A 0.000, B 0.000, C 0.000 }
gfCNCPoint2[20088] = {X 479.0692, Y 59.7984, Z -3.0000, A 0.000, B 0.000, C 0.000 }
gfCNCPoint2[20089] = {X 478.8009, Y 60.6249, Z -3.0000, A 0.000, B 0.000, C 0.000 }
gfCNCPoint2[20090] = {X 478.3667, Y 61.3776, Z -3.0000, A 0.000, B 0.000, C 0.000 }
gfCNCPoint2[20091] = {X 477.7856, Y 62.0237, Z -3.0000, A 0.000, B 0.000, C 0.000 }
gfCNCPoint2[20092] = {X 477.0830, Y 62.5350, Z -3.0000, A 0.000, B 0.000, C 0.000 }
gfCNCPoint2[20093] = {X 476.2895, Y 62.8892, Z -3.0000, A 0.000, B 0.000, C 0.000 }
gfCNCPoint2[20094] = {X 475.4397, Y 63.0708, Z -3.0000, A 0.000, B 0.000, C 0.000 }
gfCNCPoint2[20095] = {X 475.4401, Y 92.8979, Z -3.0000, A 0.000, B 0.000, C 0.000 }
gfCNCPoint2[20096] = {X 475.8916, Y 93.0049, Z -3.0000, A 0.000, B 0.000, C 0.000 }
gfCNCPoint2[20097] = {X 476.3359, Y 93.1387, Z -3.0000, A 0.000, B 0.000, C 0.000 }
gfCNCPoint2[20098] = {X 477.1176, Y 93.4938, Z -3.0000, A 0.000, B 0.000, C 0.000 }
gfCNCPoint2[20099] = {X 477.8091, Y 94.0028, Z -3.0000, A 0.000, B 0.000, C 0.000 }
gfCNCPoint2[20100] = {X 478.3805, Y 94.6435, Z -3.0000, A 0.000, B 0.000, C 0.000 }
gfCNCPoint2[20101] = {X 478.8072, Y 95.3885, Z -3.0000, A 0.000, B 0.000, C 0.000 }
gfCNCPoint2[20102] = {X 479.0708, Y 96.2056, Z -3.0000, A 0.000, B 0.000, C 0.000 }
gfCNCPoint2[20103] = {X 479.1600, Y 97.0595, Z -3.0000, A 0.000, B 0.000, C 0.000 }
gfCNCPoint2[20104] = {X 479.1600, Y 98.0000, Z -3.0000, A 0.000, B 0.000, C 0.000 }
gfCNCPoint2[20105] = {X 479.0557, Y 98.9257, Z -3.0000, A 0.000, B 0.000, C 0.000 }
gfCNCPoint2[20106] = {X 478.7480, Y 99.8050, Z -3.0000, A 0.000, B 0.000, C 0.000 }
gfCNCPoint2[20107] = {X 478.2524, Y 100.5937, Z -3.0000, A 0.000, B 0.000, C 0.000 }
gfCNCPoint2[20108] = {X 477.5937, Y 101.2524, Z -3.0000, A 0.000, B 0.000, C 0.000 }
gfCNCPoint2[20109] = {X 476.8050, Y 101.7480, Z -3.0000, A 0.000, B 0.000, C 0.000 }
gfCNCPoint2[20110] = {X 475.9257, Y 102.0557, Z -3.0000, A 0.000, B 0.000, C 0.000 }
gfCNCPoint2[20111] = {X 475.0000, Y 102.1600, Z -3.0000, A 0.000, B 0.000, C 0.000 }
gfCNCPoint2[20112] = {X 458.4596, Y 102.1600, Z -3.0000, A 0.000, B 0.000, C 0.000 }
gfCNCPoint2[20113] = {X 457.5339, Y 102.0557, Z -3.0000, A 0.000, B 0.000, C 0.000 }
gfCNCPoint2[20114] = {X 456.6546, Y 101.7480, Z -3.0000, A 0.000, B 0.000, C 0.000 }
gfCNCPoint2[20115] = {X 455.8659, Y 101.2524, Z -3.0000, A 0.000, B 0.000, C 0.000 }
gfCNCPoint2[20116] = {X 455.2072, Y 100.5937, Z -3.0000, A 0.000, B 0.000, C 0.000 }
gfCNCPoint2[20117] = {X 454.7116, Y 99.8050, Z -3.0000, A 0.000, B 0.000, C 0.000 }
gfCNCPoint2[20118] = {X 454.4039, Y 98.9257, Z -3.0000, A 0.000, B 0.000, C 0.000 }
gfCNCPoint2[20119] = {X 454.2996, Y 98.0000, Z -3.0000, A 0.000, B 0.000, C 0.000 }
gfCNCPoint2[20120] = {X 454.2996, Y 97.0659, Z -3.0000, A 0.000, B 0.000, C 0.000 }
gfCNCPoint2[20121] = {X 454.3903, Y 96.2022, Z -3.0000, A 0.000, B 0.000, C 0.000 }
gfCNCPoint2[20122] = {X 454.6583, Y 95.3761, Z -3.0000, A 0.000, B 0.000, C 0.000 }
gfCNCPoint2[20123] = {X 455.0920, Y 94.6237, Z -3.0000, A 0.000, B 0.000, C 0.000 }
gfCNCPoint2[20124] = {X 455.6724, Y 93.9777, Z -3.0000, A 0.000, B 0.000, C 0.000 }
gfCNCPoint2[20125] = {X 456.3743, Y 93.4663, Z -3.0000, A 0.000, B 0.000, C 0.000 }
gfCNCPoint2[20126] = {X 457.1672, Y 93.1118, Z -3.0000, A 0.000, B 0.000, C 0.000 }
gfCNCPoint2[20127] = {X 458.0163, Y 92.9296, Z -3.0000, A 0.000, B 0.000, C 0.000 }
gfCNCPoint2[20128] = {X 458.0163, Y 85.4858, Z -3.0000, A 0.000, B 0.000, C 0.000 }
gfCNCPoint2[20129] = {X 444.8404, Y 80.3209, Z -3.0000, A 0.000, B 0.000, C 0.000 }
gfCNCPoint2[20130] = {X 419.8623, Y 96.5016, Z -3.0000, A 0.000, B 0.000, C 0.000 }
gfCNCPoint2[20131] = {X 419.8667, Y 97.0653, Z -3.0000, A 0.000, B 0.000, C 0.000 }
gfCNCPoint2[20132] = {X 419.8667, Y 98.0000, Z -3.0000, A 0.000, B 0.000, C 0.000 }
gfCNCPoint2[20133] = {X 419.7624, Y 98.9257, Z -3.0000, A 0.000, B 0.000, C 0.000 }
gfCNCPoint2[20134] = {X 419.4547, Y 99.8050, Z -3.0000, A 0.000, B 0.000, C 0.000 }
gfCNCPoint2[20135] = {X 418.9591, Y 100.5937, Z -3.0000, A 0.000, B 0.000, C 0.000 }
gfCNCPoint2[20136] = {X 418.3004, Y 101.2524, Z -3.0000, A 0.000, B 0.000, C 0.000 }
gfCNCPoint2[20137] = {X 417.5117, Y 101.7480, Z -3.0000, A 0.000, B 0.000, C 0.000 }
gfCNCPoint2[20138] = {X 416.6324, Y 102.0557, Z -3.0000, A 0.000, B 0.000, C 0.000 }
gfCNCPoint2[20139] = {X 415.7067, Y 102.1600, Z -3.0000, A 0.000, B 0.000, C 0.000 }
gfCNCPoint2[20140] = {X 396.4059, Y 102.1600, Z -3.0000, A 0.000, B 0.000, C 0.000 }
gfCNCPoint2[20141] = {X 395.4803, Y 102.0557, Z -3.0000, A 0.000, B 0.000, C 0.000 }
gfCNCPoint2[20142] = {X 394.6010, Y 101.7480, Z -3.0000, A 0.000, B 0.000, C 0.000 }
gfCNCPoint2[20143] = {X 393.8122, Y 101.2524, Z -3.0000, A 0.000, B 0.000, C 0.000 }
gfCNCPoint2[20144] = {X 393.1535, Y 100.5937, Z -3.0000, A 0.000, B 0.000, C 0.000 }
gfCNCPoint2[20145] = {X 392.6579, Y 99.8050, Z -3.0000, A 0.000, B 0.000, C 0.000 }
gfCNCPoint2[20146] = {X 392.3502, Y 98.9257, Z -3.0000, A 0.000, B 0.000, C 0.000 }
gfCNCPoint2[20147] = {X 392.2459, Y 98.0000, Z -3.0000, A 0.000, B 0.000, C 0.000 }
gfCNCPoint2[20148] = {X 392.2459, Y 97.0659, Z -3.0000, A 0.000, B 0.000, C 0.000 }
gfCNCPoint2[20149] = {X 392.3498, Y 96.1422, Z -3.0000, A 0.000, B 0.000, C 0.000 }
gfCNCPoint2[20150] = {X 392.6562, Y 95.2646, Z -3.0000, A 0.000, B 0.000, C 0.000 }
gfCNCPoint2[20151] = {X 393.1497, Y 94.4770, Z -3.0000, A 0.000, B 0.000, C 0.000 }
gfCNCPoint2[20152] = {X 393.8059, Y 93.8186, Z -3.0000, A 0.000, B 0.000, C 0.000 }
gfCNCPoint2[20153] = {X 394.5918, Y 93.3223, Z -3.0000, A 0.000, B 0.000, C 0.000 }
gfCNCPoint2[20154] = {X 395.4684, Y 93.0130, Z -3.0000, A 0.000, B 0.000, C 0.000 }
gfCNCPoint2[20155] = {X 396.3917, Y 92.9060, Z -3.0000, A 0.000, B 0.000, C 0.000 }
gfCNCPoint2[20156] = {X 397.3541, Y 92.8649, Z -3.0000, A 0.000, B 0.000, C 0.000 }
gfCNCPoint2[20157] = {X 398.3130, Y 92.7738, Z -3.0000, A 0.000, B 0.000, C 0.000 }
gfCNCPoint2[20158] = {X 398.9990, Y 92.6076, Z -3.0000, A 0.000, B 0.000, C 0.000 }
gfCNCPoint2[20159] = {X 399.6306, Y 92.2926, Z -3.0000, A 0.000, B 0.000, C 0.000 }
gfCNCPoint2[20160] = {X 413.8857, Y 83.1636, Z -3.0000, A 0.000, B 0.000, C 0.000 }
gfCNCPoint2[20161] = {X 411.7285, Y 79.7952, Z -3.0000, A 0.000, B 0.000, C 0.000 }
gfCNCPoint2[20162] = {X 413.9288, Y 83.2310, Z -3.0000, A 0.000, B 0.000, C 0.000 }
gfCNCPoint2[20163] = {X 428.5808, Y 73.8479, Z -3.0000, A 0.000, B 0.000, C 0.000 }
gfCNCPoint2[20164] = {X 403.8433, Y 64.1418, Z -3.0000, A 0.000, B 0.000, C 0.000 }
gfCNCPoint2[20165] = {X 402.1209, Y 63.5715, Z -3.0000, A 0.000, B 0.000, C 0.000 }
gfCNCPoint2[20166] = {X 400.3462, Y 63.1941, Z -3.0000, A 0.000, B 0.000, C 0.000 }
gfCNCPoint2[20167] = {X 398.5408, Y 63.0140, Z -3.0000, A 0.000, B 0.000, C 0.000 }
gfCNCPoint2[20168] = {X 397.6404, Y 62.9096, Z -3.0000, A 0.000, B 0.000, C 0.000 }
gfCNCPoint2[20169] = {X 396.7853, Y 62.6090, Z -3.0000, A 0.000, B 0.000, C 0.000 }
gfCNCPoint2[20170] = {X 396.0177, Y 62.1270, Z -3.0000, A 0.000, B 0.000, C 0.000 }
gfCNCPoint2[20171] = {X 395.3754, Y 61.4874, Z -3.0000, A 0.000, B 0.000, C 0.000 }
gfCNCPoint2[20172] = {X 394.8902, Y 60.7217, Z -3.0000, A 0.000, B 0.000, C 0.000 }
gfCNCPoint2[20173] = {X 394.5860, Y 59.8679, Z -3.0000, A 0.000, B 0.000, C 0.000 }
gfCNCPoint2[20174] = {X 394.4779, Y 58.9680, Z -3.0000, A 0.000, B 0.000, C 0.000 }
gfCNCPoint2[20175] = {X 394.4777, Y 58.0000, Z -3.0000, A 0.000, B 0.000, C 0.000 }
gfCNCPoint2[20176] = {X 394.5800, Y 57.0921, Z -3.0000, A 0.000, B 0.000, C 0.000 }
gfCNCPoint2[20177] = {X 394.8818, Y 56.2298, Z -3.0000, A 0.000, B 0.000, C 0.000 }
gfCNCPoint2[20178] = {X 395.3679, Y 55.4562, Z -3.0000, A 0.000, B 0.000, C 0.000 }
gfCNCPoint2[20179] = {X 396.0139, Y 54.8101, Z -3.0000, A 0.000, B 0.000, C 0.000 }
gfCNCPoint2[20180] = {X 396.7875, Y 54.3240, Z -3.0000, A 0.000, B 0.000, C 0.000 }
gfCNCPoint2[20181] = {X 397.6498, Y 54.0223, Z -3.0000, A 0.000, B 0.000, C 0.000 }
gfCNCPoint2[20182] = {X 398.5577, Y 53.9200, Z -3.0000, A 0.000, B 0.000, C 0.000 }
gfCNCPoint2[20183] = {X 419.4886, Y 53.9200, Z -3.0000, A 0.000, B 0.000, C 0.000 }
gfCNCPoint2[20184] = {X 420.3965, Y 54.0223, Z -3.0000, A 0.000, B 0.000, C 0.000 }
gfCNCPoint2[20185] = {X 421.2588, Y 54.3240, Z -3.0000, A 0.000, B 0.000, C 0.000 }
gfCNCPoint2[20186] = {X 422.0324, Y 54.8101, Z -3.0000, A 0.000, B 0.000, C 0.000 }
gfCNCPoint2[20187] = {X 422.6785, Y 55.4562, Z -3.0000, A 0.000, B 0.000, C 0.000 }
gfCNCPoint2[20188] = {X 423.1646, Y 56.2298, Z -3.0000, A 0.000, B 0.000, C 0.000 }
gfCNCPoint2[20189] = {X 423.4663, Y 57.0921, Z -3.0000, A 0.000, B 0.000, C 0.000 }
gfCNCPoint2[20190] = {X 423.5686, Y 58.0000, Z -3.0000, A 0.000, B 0.000, C 0.000 }
gfCNCPoint2[20191] = {X 423.5686, Y 58.3966, Z -3.0000, A 0.000, B 0.000, C 0.000 }
gfCNCPoint2[20192] = {X 429.5238, Y 60.7174, Z -3.0000, A 0.000, B 0.000, C 0.000 }
gfCNCPoint2[20193] = {X 458.1008, Y 72.0553, Z -3.0000, A 0.000, B 0.000, C 0.000 }
gfCNCPoint2[20194] = {X 458.1011, Y 62.9983, Z -3.0000, A 0.000, B 0.000, C 0.000 }
gfCNCPoint2[20195] = {X 457.9648, Y 62.9839, Z -3.0000, A 0.000, B 0.000, C 0.000 }
gfCNCPoint2[20196] = {X 457.8290, Y 62.9650, Z -3.0000, A 0.000, B 0.000, C 0.000 }
gfCNCPoint2[20197] = {X 456.9094, Y 62.7081, Z -3.0000, A 0.000, B 0.000, C 0.000 }
gfCNCPoint2[20198] = {X 456.0747, Y 62.2445, Z -3.0000, A 0.000, B 0.000, C 0.000 }
gfCNCPoint2[20199] = {X 455.3707, Y 61.5996, Z -3.0000, A 0.000, B 0.000, C 0.000 }
gfCNCPoint2[20200] = {X 454.8357, Y 60.8086, Z -3.0000, A 0.000, B 0.000, C 0.000 }
gfCNCPoint2[20201] = {X 454.4993, Y 59.9151, Z -3.0000, A 0.000, B 0.000, C 0.000 }
gfCNCPoint2[20202] = {X 454.3797, Y 58.9678, Z -3.0000, A 0.000, B 0.000, C 0.000 }
gfCNCPoint2[20203] = {X 454.3796, Y 58.0000, Z -3.0000, A 0.000, B 0.000, C 0.000 }
gfCNCPoint2[20204] = {X 454.4819, Y 57.0921, Z -3.0000, A 0.000, B 0.000, C 0.000 }
gfCNCPoint2[20205] = {X 454.7837, Y 56.2298, Z -3.0000, A 0.000, B 0.000, C 0.000 }
gfCNCPoint2[20206] = {X 455.2697, Y 55.4562, Z -3.0000, A 0.000, B 0.000, C 0.000 }
gfCNCPoint2[20207] = {X 455.9158, Y 54.8101, Z -3.0000, A 0.000, B 0.000, C 0.000 }
gfCNCPoint2[20208] = {X 456.6894, Y 54.3240, Z -3.0000, A 0.000, B 0.000, C 0.000 }
gfCNCPoint2[20209] = {X 457.5517, Y 54.0223, Z -3.0000, A 0.000, B 0.000, C 0.000 }
gfCNCPoint2[20210] = {X 458.4596, Y 53.9200, Z -3.0000, A 0.000, B 0.000, C 0.000 }
gfCNCPoint2[20211] = {X 475.0000, Y 53.9200, Z -3.0000, A 0.000, B 0.000, C 0.000 }
gfCNCPoint2[20212] = {X 475.9079, Y 54.0223, Z -3.0000, A 0.000, B 0.000, C 0.000 }
gfCNCPoint2[20213] = {X 476.7702, Y 54.3240, Z -3.0000, A 0.000, B 0.000, C 0.000 }
gfCNCPoint2[20214] = {X 477.5438, Y 54.8101, Z -3.0000, A 0.000, B 0.000, C 0.000 }
gfCNCPoint2[20215] = {X 478.1899, Y 55.4562, Z -3.0000, A 0.000, B 0.000, C 0.000 }
gfCNCPoint2[20216] = {X 478.6760, Y 56.2298, Z -3.0000, A 0.000, B 0.000, C 0.000 }
gfCNCPoint2[20217] = {X 478.9777, Y 57.0921, Z -3.0000, A 0.000, B 0.000, C 0.000 }
gfCNCPoint2[20218] = {X 479.0800, Y 58.0000, Z -3.0000, A 0.000, B 0.000, C 0.000 }
gfCNCPoint2[20219] = {X 479.0800, Y 58.9342, Z -3.0000, A 0.000, B 0.000, C 0.000 }
gfCNCPoint2[20220] = {X 478.9888, Y 59.7918, Z -3.0000, A 0.000, B 0.000, C 0.000 }
gfCNCPoint2[20221] = {X 478.7194, Y 60.6111, Z -3.0000, A 0.000, B 0.000, C 0.000 }
gfCNCPoint2[20222] = {X 478.2838, Y 61.3555, Z -3.0000, A 0.000, B 0.000, C 0.000 }
gfCNCPoint2[20223] = {X 477.7014, Y 61.9916, Z -3.0000, A 0.000, B 0.000, C 0.000 }
gfCNCPoint2[20224] = {X 476.9983, Y 62.4912, Z -3.0000, A 0.000, B 0.000, C 0.000 }
gfCNCPoint2[20225] = {X 476.2060, Y 62.8318, Z -3.0000, A 0.000, B 0.000, C 0.000 }
gfCNCPoint2[20226] = {X 475.3597, Y 62.9982, Z -3.0000, A 0.000, B 0.000, C 0.000 }
gfCNCPoint2[20227] = {X 475.3601, Y 92.9635, Z -3.0000, A 0.000, B 0.000, C 0.000 }
gfCNCPoint2[20228] = {X 475.8394, Y 93.0738, Z -3.0000, A 0.000, B 0.000, C 0.000 }
gfCNCPoint2[20229] = {X 476.3106, Y 93.2146, Z -3.0000, A 0.000, B 0.000, C 0.000 }
gfCNCPoint2[20230] = {X 477.0771, Y 93.5628, Z -3.0000, A 0.000, B 0.000, C 0.000 }
gfCNCPoint2[20231] = {X 477.7552, Y 94.0619, Z -3.0000, A 0.000, B 0.000, C 0.000 }
gfCNCPoint2[20232] = {X 478.3156, Y 94.6903, Z -3.0000, A 0.000, B 0.000, C 0.000 }
gfCNCPoint2[20233] = {X 478.7340, Y 95.4209, Z -3.0000, A 0.000, B 0.000, C 0.000 }
gfCNCPoint2[20234] = {X 478.9926, Y 96.2222, Z -3.0000, A 0.000, B 0.000, C 0.000 }
gfCNCPoint2[20235] = {X 479.0800, Y 97.0595, Z -3.0000, A 0.000, B 0.000, C 0.000 }
gfCNCPoint2[20236] = {X 479.0800, Y 98.0000, Z -3.0000, A 0.000, B 0.000, C 0.000 }
gfCNCPoint2[20237] = {X 478.9777, Y 98.9079, Z -3.0000, A 0.000, B 0.000, C 0.000 }
gfCNCPoint2[20238] = {X 478.6760, Y 99.7702, Z -3.0000, A 0.000, B 0.000, C 0.000 }
gfCNCPoint2[20239] = {X 478.1899, Y 100.5438, Z -3.0000, A 0.000, B 0.000, C 0.000 }
gfCNCPoint2[20240] = {X 477.5438, Y 101.1899, Z -3.0000, A 0.000, B 0.000, C 0.000 }
gfCNCPoint2[20241] = {X 476.7702, Y 101.6760, Z -3.0000, A 0.000, B 0.000, C 0.000 }
gfCNCPoint2[20242] = {X 475.9079, Y 101.9777, Z -3.0000, A 0.000, B 0.000, C 0.000 }
gfCNCPoint2[20243] = {X 475.0000, Y 102.0800, Z -3.0000, A 0.000, B 0.000, C 0.000 }
gfCNCPoint2[20244] = {X 458.4596, Y 102.0800, Z -3.0000, A 0.000, B 0.000, C 0.000 }
gfCNCPoint2[20245] = {X 457.5517, Y 101.9777, Z -3.0000, A 0.000, B 0.000, C 0.000 }
gfCNCPoint2[20246] = {X 456.6894, Y 101.6760, Z -3.0000, A 0.000, B 0.000, C 0.000 }
gfCNCPoint2[20247] = {X 455.9158, Y 101.1899, Z -3.0000, A 0.000, B 0.000, C 0.000 }
gfCNCPoint2[20248] = {X 455.2697, Y 100.5438, Z -3.0000, A 0.000, B 0.000, C 0.000 }
gfCNCPoint2[20249] = {X 454.7837, Y 99.7702, Z -3.0000, A 0.000, B 0.000, C 0.000 }
gfCNCPoint2[20250] = {X 454.4819, Y 98.9079, Z -3.0000, A 0.000, B 0.000, C 0.000 }
gfCNCPoint2[20251] = {X 454.3796, Y 98.0000, Z -3.0000, A 0.000, B 0.000, C 0.000 }
gfCNCPoint2[20252] = {X 454.3796, Y 97.0659, Z -3.0000, A 0.000, B 0.000, C 0.000 }
gfCNCPoint2[20253] = {X 454.4707, Y 96.2088, Z -3.0000, A 0.000, B 0.000, C 0.000 }
gfCNCPoint2[20254] = {X 454.7398, Y 95.3899, Z -3.0000, A 0.000, B 0.000, C 0.000 }
gfCNCPoint2[20255] = {X 455.1749, Y 94.6458, Z -3.0000, A 0.000, B 0.000, C 0.000 }
gfCNCPoint2[20256] = {X 455.7566, Y 94.0098, Z -3.0000, A 0.000, B 0.000, C 0.000 }
gfCNCPoint2[20257] = {X 456.4590, Y 93.5101, Z -3.0000, A 0.000, B 0.000, C 0.000 }
gfCNCPoint2[20258] = {X 457.2507, Y 93.1692, Z -3.0000, A 0.000, B 0.000, C 0.000 }
gfCNCPoint2[20259] = {X 458.0963, Y 93.0021, Z -3.0000, A 0.000, B 0.000, C 0.000 }
gfCNCPoint2[20260] = {X 458.0963, Y 85.4313, Z -3.0000, A 0.000, B 0.000, C 0.000 }
gfCNCPoint2[20261] = {X 444.8314, Y 80.2314, Z -3.0000, A 0.000, B 0.000, C 0.000 }
gfCNCPoint2[20262] = {X 419.7819, Y 96.4583, Z -3.0000, A 0.000, B 0.000, C 0.000 }
gfCNCPoint2[20263] = {X 419.7867, Y 97.0656, Z -3.0000, A 0.000, B 0.000, C 0.000 }
gfCNCPoint2[20264] = {X 419.7867, Y 98.0000, Z -3.0000, A 0.000, B 0.000, C 0.000 }
gfCNCPoint2[20265] = {X 419.6844, Y 98.9079, Z -3.0000, A 0.000, B 0.000, C 0.000 }
gfCNCPoint2[20266] = {X 419.3827, Y 99.7702, Z -3.0000, A 0.000, B 0.000, C 0.000 }
gfCNCPoint2[20267] = {X 418.8966, Y 100.5438, Z -3.0000, A 0.000, B 0.000, C 0.000 }
gfCNCPoint2[20268] = {X 418.2505, Y 101.1899, Z -3.0000, A 0.000, B 0.000, C 0.000 }
gfCNCPoint2[20269] = {X 417.4769, Y 101.6760, Z -3.0000, A 0.000, B 0.000, C 0.000 }
gfCNCPoint2[20270] = {X 416.6146, Y 101.9777, Z -3.0000, A 0.000, B 0.000, C 0.000 }
gfCNCPoint2[20271] = {X 415.7067, Y 102.0800, Z -3.0000, A 0.000, B 0.000, C 0.000 }
gfCNCPoint2[20272] = {X 396.4059, Y 102.0800, Z -3.0000, A 0.000, B 0.000, C 0.000 }
gfCNCPoint2[20273] = {X 395.4981, Y 101.9777, Z -3.0000, A 0.000, B 0.000, C 0.000 }
gfCNCPoint2[20274] = {X 394.6357, Y 101.6760, Z -3.0000, A 0.000, B 0.000, C 0.000 }
gfCNCPoint2[20275] = {X 393.8621, Y 101.1899, Z -3.0000, A 0.000, B 0.000, C 0.000 }
gfCNCPoint2[20276] = {X 393.2161, Y 100.5438, Z -3.0000, A 0.000, B 0.000, C 0.000 }
gfCNCPoint2[20277] = {X 392.7300, Y 99.7702, Z -3.0000, A 0.000, B 0.000, C 0.000 }
gfCNCPoint2[20278] = {X 392.4282, Y 98.9079, Z -3.0000, A 0.000, B 0.000, C 0.000 }
gfCNCPoint2[20279] = {X 392.3259, Y 98.0000, Z -3.0000, A 0.000, B 0.000, C 0.000 }
gfCNCPoint2[20280] = {X 392.3259, Y 97.0659, Z -3.0000, A 0.000, B 0.000, C 0.000 }
gfCNCPoint2[20281] = {X 392.4278, Y 96.1599, Z -3.0000, A 0.000, B 0.000, C 0.000 }
gfCNCPoint2[20282] = {X 392.7283, Y 95.2991, Z -3.0000, A 0.000, B 0.000, C 0.000 }
gfCNCPoint2[20283] = {X 393.2125, Y 94.5266, Z -3.0000, A 0.000, B 0.000, C 0.000 }
gfCNCPoint2[20284] = {X 393.8561, Y 93.8809, Z -3.0000, A 0.000, B 0.000, C 0.000 }
gfCNCPoint2[20285] = {X 394.6271, Y 93.3942, Z -3.0000, A 0.000, B 0.000, C 0.000 }
gfCNCPoint2[20286] = {X 395.4868, Y 93.0908, Z -3.0000, A 0.000, B 0.000, C 0.000 }
gfCNCPoint2[20287] = {X 396.3925, Y 92.9860, Z -3.0000, A 0.000, B 0.000, C 0.000 }
gfCNCPoint2[20288] = {X 397.3594, Y 92.9447, Z -3.0000, A 0.000, B 0.000, C 0.000 }
gfCNCPoint2[20289] = {X 398.3229, Y 92.8532, Z -3.0000, A 0.000, B 0.000, C 0.000 }
gfCNCPoint2[20290] = {X 399.0264, Y 92.6828, Z -3.0000, A 0.000, B 0.000, C 0.000 }
gfCNCPoint2[20291] = {X 399.6742, Y 92.3597, Z -3.0000, A 0.000, B 0.000, C 0.000 }
gfCNCPoint2[20292] = {X 413.9288, Y 83.2310, Z -3.0000, A 0.000, B 0.000, C 0.000 }
gfCNCPoint2[20293] = {X 411.7651, Y 79.8524, Z -3.0000, A 0.000, B 0.000, C 0.000 }
gfCNCPoint2[20294] = {X 411.7675, Y 79.8509, Z -3.0000, A 0.000, B 0.000, C 0.000 }
gfCNCPoint2[20295] = {X 413.9654, Y 83.2883, Z -3.0000, A 0.000, B 0.000, C 0.000 }
gfCNCPoint2[20296] = {X 428.7561, Y 73.8307, Z -3.0000, A 0.000, B 0.000, C 0.000 }
gfCNCPoint2[20297] = {X 403.8726, Y 64.0674, Z -3.0000, A 0.000, B 0.000, C 0.000 }
gfCNCPoint2[20298] = {X 402.1413, Y 63.4942, Z -3.0000, A 0.000, B 0.000, C 0.000 }
gfCNCPoint2[20299] = {X 400.3575, Y 63.1149, Z -3.0000, A 0.000, B 0.000, C 0.000 }
gfCNCPoint2[20300] = {X 398.5427, Y 62.9340, Z -3.0000, A 0.000, B 0.000, C 0.000 }
gfCNCPoint2[20301] = {X 397.6551, Y 62.8309, Z -3.0000, A 0.000, B 0.000, C 0.000 }
gfCNCPoint2[20302] = {X 396.8125, Y 62.5333, Z -3.0000, A 0.000, B 0.000, C 0.000 }
gfCNCPoint2[20303] = {X 396.0571, Y 62.0560, Z -3.0000, A 0.000, B 0.000, C 0.000 }
gfCNCPoint2[20304] = {X 395.4264, Y 61.4230, Z -3.0000, A 0.000, B 0.000, C 0.000 }
gfCNCPoint2[20305] = {X 394.9520, Y 60.6657, Z -3.0000, A 0.000, B 0.000, C 0.000 }
gfCNCPoint2[20306] = {X 394.6575, Y 59.8220, Z -3.0000, A 0.000, B 0.000, C 0.000 }
gfCNCPoint2[20307] = {X 394.5577, Y 58.9340, Z -3.0000, A 0.000, B 0.000, C 0.000 }
gfCNCPoint2[20308] = {X 394.5577, Y 58.0000, Z -3.0000, A 0.000, B 0.000, C 0.000 }
gfCNCPoint2[20309] = {X 394.6580, Y 57.1099, Z -3.0000, A 0.000, B 0.000, C 0.000 }
gfCNCPoint2[20310] = {X 394.9538, Y 56.2645, Z -3.0000, A 0.000, B 0.000, C 0.000 }
gfCNCPoint2[20311] = {X 395.4304, Y 55.5060, Z -3.0000, A 0.000, B 0.000, C 0.000 }
gfCNCPoint2[20312] = {X 396.0638, Y 54.8727, Z -3.0000, A 0.000, B 0.000, C 0.000 }
gfCNCPoint2[20313] = {X 396.8222, Y 54.3961, Z -3.0000, A 0.000, B 0.000, C 0.000 }
gfCNCPoint2[20314] = {X 397.6676, Y 54.1003, Z -3.0000, A 0.000, B 0.000, C 0.000 }
gfCNCPoint2[20315] = {X 398.5577, Y 54.0000, Z -3.0000, A 0.000, B 0.000, C 0.000 }
gfCNCPoint2[20316] = {X 419.4886, Y 54.0000, Z -3.0000, A 0.000, B 0.000, C 0.000 }
gfCNCPoint2[20317] = {X 420.3787, Y 54.1003, Z -3.0000, A 0.000, B 0.000, C 0.000 }
gfCNCPoint2[20318] = {X 421.2241, Y 54.3961, Z -3.0000, A 0.000, B 0.000, C 0.000 }
gfCNCPoint2[20319] = {X 421.9826, Y 54.8727, Z -3.0000, A 0.000, B 0.000, C 0.000 }
gfCNCPoint2[20320] = {X 422.6159, Y 55.5060, Z -3.0000, A 0.000, B 0.000, C 0.000 }
gfCNCPoint2[20321] = {X 423.0925, Y 56.2645, Z -3.0000, A 0.000, B 0.000, C 0.000 }
gfCNCPoint2[20322] = {X 423.3883, Y 57.1099, Z -3.0000, A 0.000, B 0.000, C 0.000 }
gfCNCPoint2[20323] = {X 423.4886, Y 58.0000, Z -3.0000, A 0.000, B 0.000, C 0.000 }
gfCNCPoint2[20324] = {X 423.4886, Y 58.4513, Z -3.0000, A 0.000, B 0.000, C 0.000 }
gfCNCPoint2[20325] = {X 429.4945, Y 60.7918, Z -3.0000, A 0.000, B 0.000, C 0.000 }
gfCNCPoint2[20326] = {X 458.1789, Y 72.1724, Z -3.0000, A 0.000, B 0.000, C 0.000 }
gfCNCPoint2[20327] = {X 458.1807, Y 71.5840, Z -3.0000, A 0.000, B 0.000, C 0.000 }
gfCNCPoint2[20328] = {X 458.1796, Y 63.0382, Z -3.0000, A 0.000, B 0.000, C 0.000 }
gfCNCPoint2[20329] = {X 458.1841, Y 62.9246, Z -3.0000, A 0.000, B 0.000, C 0.000 }
gfCNCPoint2[20330] = {X 458.0123, Y 62.9090, Z -3.0000, A 0.000, B 0.000, C 0.000 }
gfCNCPoint2[20331] = {X 457.8414, Y 62.8860, Z -3.0000, A 0.000, B 0.000, C 0.000 }
gfCNCPoint2[20332] = {X 456.9347, Y 62.6320, Z -3.0000, A 0.000, B 0.000, C 0.000 }
gfCNCPoint2[20333] = {X 456.1126, Y 62.1731, Z -3.0000, A 0.000, B 0.000, C 0.000 }
gfCNCPoint2[20334] = {X 455.4205, Y 61.5348, Z -3.0000, A 0.000, B 0.000, C 0.000 }
gfCNCPoint2[20335] = {X 454.8967, Y 60.7523, Z -3.0000, A 0.000, B 0.000, C 0.000 }
gfCNCPoint2[20336] = {X 454.5704, Y 59.8691, Z -3.0000, A 0.000, B 0.000, C 0.000 }
gfCNCPoint2[20337] = {X 454.4596, Y 58.9340, Z -3.0000, A 0.000, B 0.000, C 0.000 }
gfCNCPoint2[20338] = {X 454.4596, Y 58.0000, Z -3.0000, A 0.000, B 0.000, C 0.000 }
gfCNCPoint2[20339] = {X 454.5599, Y 57.1099, Z -3.0000, A 0.000, B 0.000, C 0.000 }
gfCNCPoint2[20340] = {X 454.8557, Y 56.2645, Z -3.0000, A 0.000, B 0.000, C 0.000 }
gfCNCPoint2[20341] = {X 455.3323, Y 55.5060, Z -3.0000, A 0.000, B 0.000, C 0.000 }
gfCNCPoint2[20342] = {X 455.9656, Y 54.8727, Z -3.0000, A 0.000, B 0.000, C 0.000 }
gfCNCPoint2[20343] = {X 456.7241, Y 54.3961, Z -3.0000, A 0.000, B 0.000, C 0.000 }
gfCNCPoint2[20344] = {X 457.5695, Y 54.1003, Z -3.0000, A 0.000, B 0.000, C 0.000 }
gfCNCPoint2[20345] = {X 458.4596, Y 54.0000, Z -3.0000, A 0.000, B 0.000, C 0.000 }
gfCNCPoint2[20346] = {X 475.0000, Y 54.0000, Z -3.0000, A 0.000, B 0.000, C 0.000 }
gfCNCPoint2[20347] = {X 475.8901, Y 54.1003, Z -3.0000, A 0.000, B 0.000, C 0.000 }
gfCNCPoint2[20348] = {X 476.7355, Y 54.3961, Z -3.0000, A 0.000, B 0.000, C 0.000 }
gfCNCPoint2[20349] = {X 477.4940, Y 54.8727, Z -3.0000, A 0.000, B 0.000, C 0.000 }
gfCNCPoint2[20350] = {X 478.1273, Y 55.5060, Z -3.0000, A 0.000, B 0.000, C 0.000 }
gfCNCPoint2[20351] = {X 478.6039, Y 56.2645, Z -3.0000, A 0.000, B 0.000, C 0.000 }
gfCNCPoint2[20352] = {X 478.8997, Y 57.1099, Z -3.0000, A 0.000, B 0.000, C 0.000 }
gfCNCPoint2[20353] = {X 479.0000, Y 58.0000, Z -3.0000, A 0.000, B 0.000, C 0.000 }
gfCNCPoint2[20354] = {X 478.9999, Y 58.9671, Z -3.0000, A 0.000, B 0.000, C 0.000 }
gfCNCPoint2[20355] = {X 478.9023, Y 59.8128, Z -3.0000, A 0.000, B 0.000, C 0.000 }
gfCNCPoint2[20356] = {X 478.6280, Y 60.6186, Z -3.0000, A 0.000, B 0.000, C 0.000 }
gfCNCPoint2[20357] = {X 478.1894, Y 61.3482, Z -3.0000, A 0.000, B 0.000, C 0.000 }
gfCNCPoint2[20358] = {X 477.6063, Y 61.9684, Z -3.0000, A 0.000, B 0.000, C 0.000 }
gfCNCPoint2[20359] = {X 476.9052, Y 62.4512, Z -3.0000, A 0.000, B 0.000, C 0.000 }
gfCNCPoint2[20360] = {X 476.1177, Y 62.7747, Z -3.0000, A 0.000, B 0.000, C 0.000 }
gfCNCPoint2[20361] = {X 475.2797, Y 62.9243, Z -3.0000, A 0.000, B 0.000, C 0.000 }
gfCNCPoint2[20362] = {X 475.2801, Y 93.0295, Z -3.0000, A 0.000, B 0.000, C 0.000 }
gfCNCPoint2[20363] = {X 475.7872, Y 93.1428, Z -3.0000, A 0.000, B 0.000, C 0.000 }
gfCNCPoint2[20364] = {X 476.2852, Y 93.2905, Z -3.0000, A 0.000, B 0.000, C 0.000 }
gfCNCPoint2[20365] = {X 477.0367, Y 93.6319, Z -3.0000, A 0.000, B 0.000, C 0.000 }
gfCNCPoint2[20366] = {X 477.7014, Y 94.1211, Z -3.0000, A 0.000, B 0.000, C 0.000 }
gfCNCPoint2[20367] = {X 478.2507, Y 94.7371, Z -3.0000, A 0.000, B 0.000, C 0.000 }
gfCNCPoint2[20368] = {X 478.6609, Y 95.4532, Z -3.0000, A 0.000, B 0.000, C 0.000 }
gfCNCPoint2[20369] = {X 478.9143, Y 96.2387, Z -3.0000, A 0.000, B 0.000, C 0.000 }
gfCNCPoint2[20370] = {X 479.0000, Y 97.0595, Z -3.0000, A 0.000, B 0.000, C 0.000 }
gfCNCPoint2[20371] = {X 479.0000, Y 98.0000, Z -3.0000, A 0.000, B 0.000, C 0.000 }
gfCNCPoint2[20372] = {X 478.8997, Y 98.8901, Z -3.0000, A 0.000, B 0.000, C 0.000 }
gfCNCPoint2[20373] = {X 478.6039, Y 99.7355, Z -3.0000, A 0.000, B 0.000, C 0.000 }
gfCNCPoint2[20374] = {X 478.1273, Y 100.4940, Z -3.0000, A 0.000, B 0.000, C 0.000 }
gfCNCPoint2[20375] = {X 477.4940, Y 101.1273, Z -3.0000, A 0.000, B 0.000, C 0.000 }
gfCNCPoint2[20376] = {X 476.7355, Y 101.6039, Z -3.0000, A 0.000, B 0.000, C 0.000 }
gfCNCPoint2[20377] = {X 475.8901, Y 101.8997, Z -3.0000, A 0.000, B 0.000, C 0.000 }
gfCNCPoint2[20378] = {X 475.0000, Y 102.0000, Z -3.0000, A 0.000, B 0.000, C 0.000 }
gfCNCPoint2[20379] = {X 458.4596, Y 102.0000, Z -3.0000, A 0.000, B 0.000, C 0.000 }
gfCNCPoint2[20380] = {X 457.5695, Y 101.8997, Z -3.0000, A 0.000, B 0.000, C 0.000 }
gfCNCPoint2[20381] = {X 456.7241, Y 101.6039, Z -3.0000, A 0.000, B 0.000, C 0.000 }
gfCNCPoint2[20382] = {X 455.9656, Y 101.1273, Z -3.0000, A 0.000, B 0.000, C 0.000 }
gfCNCPoint2[20383] = {X 455.3323, Y 100.4940, Z -3.0000, A 0.000, B 0.000, C 0.000 }
gfCNCPoint2[20384] = {X 454.8557, Y 99.7355, Z -3.0000, A 0.000, B 0.000, C 0.000 }
gfCNCPoint2[20385] = {X 454.5599, Y 98.8901, Z -3.0000, A 0.000, B 0.000, C 0.000 }
gfCNCPoint2[20386] = {X 454.4596, Y 98.0000, Z -3.0000, A 0.000, B 0.000, C 0.000 }
gfCNCPoint2[20387] = {X 454.4596, Y 97.0659, Z -3.0000, A 0.000, B 0.000, C 0.000 }
gfCNCPoint2[20388] = {X 454.5511, Y 96.2154, Z -3.0000, A 0.000, B 0.000, C 0.000 }
gfCNCPoint2[20389] = {X 454.8213, Y 95.4037, Z -3.0000, A 0.000, B 0.000, C 0.000 }
gfCNCPoint2[20390] = {X 455.2580, Y 94.6681, Z -3.0000, A 0.000, B 0.000, C 0.000 }
gfCNCPoint2[20391] = {X 455.8411, Y 94.0422, Z -3.0000, A 0.000, B 0.000, C 0.000 }
gfCNCPoint2[20392] = {X 456.5439, Y 93.5545, Z -3.0000, A 0.000, B 0.000, C 0.000 }
gfCNCPoint2[20393] = {X 457.3344, Y 93.2275, Z -3.0000, A 0.000, B 0.000, C 0.000 }
gfCNCPoint2[20394] = {X 458.1763, Y 93.0760, Z -3.0000, A 0.000, B 0.000, C 0.000 }
gfCNCPoint2[20395] = {X 458.1763, Y 85.3767, Z -3.0000, A 0.000, B 0.000, C 0.000 }
gfCNCPoint2[20396] = {X 445.0135, Y 80.2169, Z -3.0000, A 0.000, B 0.000, C 0.000 }
gfCNCPoint2[20397] = {X 444.8193, Y 80.1439, Z -3.0000, A 0.000, B 0.000, C 0.000 }
gfCNCPoint2[20398] = {X 419.7016, Y 96.4150, Z -3.0000, A 0.000, B 0.000, C 0.000 }
gfCNCPoint2[20399] = {X 419.7067, Y 97.0659, Z -3.0000, A 0.000, B 0.000, C 0.000 }
gfCNCPoint2[20400] = {X 419.7067, Y 98.0000, Z -3.0000, A 0.000, B 0.000, C 0.000 }
gfCNCPoint2[20401] = {X 419.6064, Y 98.8901, Z -3.0000, A 0.000, B 0.000, C 0.000 }
gfCNCPoint2[20402] = {X 419.3106, Y 99.7355, Z -3.0000, A 0.000, B 0.000, C 0.000 }
gfCNCPoint2[20403] = {X 418.8340, Y 100.4940, Z -3.0000, A 0.000, B 0.000, C 0.000 }
gfCNCPoint2[20404] = {X 418.2007, Y 101.1273, Z -3.0000, A 0.000, B 0.000, C 0.000 }
gfCNCPoint2[20405] = {X 417.4422, Y 101.6039, Z -3.0000, A 0.000, B 0.000, C 0.000 }
gfCNCPoint2[20406] = {X 416.5968, Y 101.8997, Z -3.0000, A 0.000, B 0.000, C 0.000 }
gfCNCPoint2[20407] = {X 415.7067, Y 102.0000, Z -3.0000, A 0.000, B 0.000, C 0.000 }
gfCNCPoint2[20408] = {X 396.4059, Y 102.0000, Z -3.0000, A 0.000, B 0.000, C 0.000 }
gfCNCPoint2[20409] = {X 395.5159, Y 101.8997, Z -3.0000, A 0.000, B 0.000, C 0.000 }
gfCNCPoint2[20410] = {X 394.6704, Y 101.6039, Z -3.0000, A 0.000, B 0.000, C 0.000 }
